; move to the rack
TRIGGER WHEN DISTANCE=1 DELAY=-1 DO Schrittmerker_R1Place(10310,10002,FPlace_R1_L4_S4_VP1,XPlace_R1_L4_S4_VP1) PRIO=-1
;FOLD PTP Place_R1_L4_S4_VP1 CONT Vel=12 % PPlace_R1_L4_S4_VP1 Tool[2]:Lower Gripper Base[0];%{PE}%R8.3.21,%MKUKATPBASIS,%CMOVE,%VPTP,%P 1:PTP, 2:Place_R1_L4_S4_VP1, 3:C_DIS, 5:12, 7:PPlace_R1_L4_S4_VP1
$BWDSTART=FALSE
PDAT_ACT= PPPlace_R1_L4_S4_VP1
FDAT_ACT= FPlace_R1_L4_S4_VP1
BAS(#PTP_PARAMS,12)
PTP XPlace_R1_L4_S4_VP1 C_DIS
;ENDFOLD
TRIGGER WHEN DISTANCE=1 DELAY=-1 DO Schrittmerker_R1Place(10311,10310,FPlace_R1_L4_S4_VP2,XPlace_R1_L4_S4_VP2) PRIO=-1
;FOLD PTP Place_R1_L4_S4_VP2 CONT Vel=12 % PPlace_R1_L4_S4_VP2 Tool[2]:Lower Gripper Base[0];%{PE}%R8.3.21,%MKUKATPBASIS,%CMOVE,%VPTP,%P 1:PTP, 2:Place_R1_L4_S4_VP2, 3:C_DIS, 5:12, 7:PPlace_R1_L4_S4_VP2
$BWDSTART=FALSE
PDAT_ACT= PPPlace_R1_L4_S4_VP2
FDAT_ACT= FPlace_R1_L4_S4_VP2
BAS(#PTP_PARAMS,12)
PTP XPlace_R1_L4_S4_VP2 C_DIS
;ENDFOLD
TRIGGER WHEN DISTANCE=1 DELAY=-1 DO Schrittmerker_R1Place(10312,10311,FPlace_R1_L4_S4_VP3,XPlace_R1_L4_S4_VP3) PRIO=-1
;FOLD PTP Place_R1_L4_S4_VP3 CONT Vel=12 % PPlace_R1_L4_S4_VP3 Tool[2]:Lower Gripper Base[1]:Rack1;%{PE}%R8.3.21,%MKUKATPBASIS,%CMOVE,%VPTP,%P 1:PTP, 2:Place_R1_L4_S4_VP3, 3:C_DIS, 5:12, 7:PPlace_R1_L4_S4_VP3
$BWDSTART=FALSE
PDAT_ACT= PPPlace_R1_L4_S4_VP3
FDAT_ACT= FPlace_R1_L4_S4_VP3
BAS(#PTP_PARAMS,12)
PTP XPlace_R1_L4_S4_VP3 C_DIS
;ENDFOLD

TRIGGER WHEN DISTANCE=1 DELAY=-1 DO Schrittmerker_R1Place(10313,10312,FPlace_R1_L4_S4_Check,XPlace_R1_L4_S4_Check) PRIO=-1
;FOLD PTP Place_R1_L4_S4_Check Vel=12 % PPlace_R1_L4_S4_Check Tool[2]:Lower Gripper Base[1]:Rack1;%{PE}%R8.3.21,%MKUKATPBASIS,%CMOVE,%VPTP,%P 1:PTP, 2:Place_R1_L4_S4_Check, 3:, 5:12, 7:PPlace_R1_L4_S4_Check
$BWDSTART=FALSE
PDAT_ACT= PPPlace_R1_L4_S4_Check
FDAT_ACT= FPlace_R1_L4_S4_Check
BAS(#PTP_PARAMS,12)
PTP XPlace_R1_L4_S4_Check
;ENDFOLD

;***************************************************
;FOLD Pruefe Platz frei
IF (DetectPart(CHECK_SHELF,PLACE)==OCCUPIED) THEN
  UP_Rueckzug_R1Place( )
  RETURN
ENDIF
;ENDFOLD
;***************************************************

TRIGGER WHEN DISTANCE=1 DELAY=-1 DO Schrittmerker_R1Place(10314,10313,FPlace_R1_L4_S4_VP4,XPlace_R1_L4_S4_VP4) PRIO=-1
;FOLD LIN Place_R1_L4_S4_VP4 CONT Vel=0.5 m/s LPlace_R1_L4_S4_VP4 Tool[2]:Lower Gripper Base[1]:Rack1;%{PE}%R8.3.21,%MKUKATPBASIS,%CMOVE,%VLIN,%P 1:LIN, 2:Place_R1_L4_S4_VP4, 3:C_DIS C_DIS, 5:0.5, 7:LPlace_R1_L4_S4_VP4
$BWDSTART=FALSE
LDAT_ACT= LLPlace_R1_L4_S4_VP4
FDAT_ACT= FPlace_R1_L4_S4_VP4
BAS(#CP_PARAMS,0.5)
LIN XPlace_R1_L4_S4_VP4 C_DIS C_DIS
;ENDFOLD
TRIGGER WHEN DISTANCE=1 DELAY=-1 DO Schrittmerker_R1Place(10315,10314,FPlace_R1_L4_S4_VP5,XPlace_R1_L4_S4_VP5) PRIO=-1
;FOLD LIN Place_R1_L4_S4_VP5 CONT Vel=0.5 m/s LPlace_R1_L4_S4_VP5 Tool[2]:Lower Gripper Base[1]:Rack1;%{PE}%R8.3.21,%MKUKATPBASIS,%CMOVE,%VLIN,%P 1:LIN, 2:Place_R1_L4_S4_VP5, 3:C_DIS C_DIS, 5:0.5, 7:LPlace_R1_L4_S4_VP5
$BWDSTART=FALSE
LDAT_ACT= LLPlace_R1_L4_S4_VP5
FDAT_ACT= FPlace_R1_L4_S4_VP5
BAS(#CP_PARAMS,0.5)
LIN XPlace_R1_L4_S4_VP5 C_DIS C_DIS
;ENDFOLD

;FOLD Test the way back home - part 1
CONTINUE
IF ($FLAG[M_Test_GrdstFahren1] AND NOT $FLAG[M_Test_GrdstFahren2]) THEN
  $FLAG[M_Test_GrdstFahren2]=TRUE
  UP_Rueckzug( )
  RETURN
ENDIF
;ENDFOLD

;-------------------------------
; Place part position
;-------------------------------
TRIGGER WHEN DISTANCE=1 DELAY=-1 DO Schrittmerker_R1Place(10316,10317,FPlace_R1_L4_S4_AP,XPlace_R1_L4_S4_AP) PRIO=-1
;FOLD LIN Place_R1_L4_S4_AP Vel=0.2 m/s LPlace_R1_L4_S4_AP Tool[2]:Lower Gripper Base[1]:Rack1;%{PE}%R8.3.21,%MKUKATPBASIS,%CMOVE,%VLIN,%P 1:LIN, 2:Place_R1_L4_S4_AP, 3:, 5:0.2, 7:LPlace_R1_L4_S4_AP
$BWDSTART=FALSE
LDAT_ACT= LLPlace_R1_L4_S4_AP
FDAT_ACT= FPlace_R1_L4_S4_AP
BAS(#CP_PARAMS,0.2)
LIN XPlace_R1_L4_S4_AP
;ENDFOLD

;FOLD Test the way back home - part 2
CONTINUE
IF $FLAG[M_Test_GrdstFahren2] THEN
  $FLAG[M_Test_GrdstFahren2]=FALSE
  UP_Rueckzug( )
  RETURN
ENDIF
;ENDFOLD

;***************************************************
; Disable part lost detection
SetPartLostDetection(NO_PART)
;***************************************************

TRIGGER WHEN DISTANCE=1 DELAY=-1 DO Schrittmerker_R1Place(10317,10318,FPlace_R1_L4_S4_NP1,XPlace_R1_L4_S4_NP1) PRIO=-1
;FOLD LIN Place_R1_L4_S4_NP1 Vel=0.2 m/s LPlace_R1_L4_S4_NP1 Tool[2]:Lower Gripper Base[1]:Rack1;%{PE}%R8.3.21,%MKUKATPBASIS,%CMOVE,%VLIN,%P 1:LIN, 2:Place_R1_L4_S4_NP1, 3:C_DIS C_DIS, 5:0.2, 7:LPlace_R1_L4_S4_NP1
$BWDSTART=FALSE
LDAT_ACT= LLPlace_R1_L4_S4_NP1
FDAT_ACT= FPlace_R1_L4_S4_NP1
BAS(#CP_PARAMS,0.2)
LIN XPlace_R1_L4_S4_NP1
;ENDFOLD

;***************************************************
; Check for part present (empty gripper)
CheckPartPresent(EMPTY_GRIPPER)
;***************************************************
; set load data
SetLoadData( )
;***************************************************

TRIGGER WHEN DISTANCE=1 DELAY=-1 DO Schrittmerker_R1Place(10318,10319,FPlace_R1_L4_S4_NP2,XPlace_R1_L4_S4_NP2) PRIO=-1
;FOLD LIN Place_R1_L4_S4_NP2 CONT Vel=0.5 m/s LPlace_R1_L4_S4_NP2 Tool[2]:Lower Gripper Base[1]:Rack1;%{PE}%R8.3.21,%MKUKATPBASIS,%CMOVE,%VLIN,%P 1:LIN, 2:Place_R1_L4_S4_NP2, 3:C_DIS C_DIS, 5:0.5, 7:LPlace_R1_L4_S4_NP2
$BWDSTART=FALSE
LDAT_ACT= LLPlace_R1_L4_S4_NP2
FDAT_ACT= FPlace_R1_L4_S4_NP2
BAS(#CP_PARAMS,0.5)
LIN XPlace_R1_L4_S4_NP2 C_DIS C_DIS
;ENDFOLD
TRIGGER WHEN DISTANCE=1 DELAY=-1 DO Schrittmerker_R1Place(10319,10320,FPlace_R1_L4_S4_NP3,XPlace_R1_L4_S4_NP3) PRIO=-1
;FOLD LIN Place_R1_L4_S4_NP3 Vel=0.5 m/s LPlace_R1_L4_S4_NP3 Tool[2]:Lower Gripper Base[1]:Rack 1 ;%{PE}
$BWDSTART=FALSE
LDAT_ACT= LLPlace_R1_L4_S4_NP3
FDAT_ACT= FPlace_R1_L4_S4_NP3
BAS(#CP_PARAMS,0.5)
LIN XPlace_R1_L4_S4_NP3
;ENDFOLD
TRIGGER WHEN DISTANCE=1 DELAY=-1 DO Schrittmerker_R1Place(10320,10321,FPlace_R1_L4_S4_NP4,XPlace_R1_L4_S4_NP4) PRIO=-1
;FOLD PTP Place_R1_L4_S4_NP4 CONT Vel=100 % PPlace_R1_L4_S4_NP4 Tool[2]:Lower Gripper Base[0];%{PE}%R8.3.21,%MKUKATPBASIS,%CMOVE,%VPTP,%P 1:PTP, 2:Place_R1_L4_S4_NP4, 3:C_DIS, 5:100, 7:PPlace_R1_L4_S4_NP4
$BWDSTART=FALSE
PDAT_ACT= PPPlace_R1_L4_S4_NP4
FDAT_ACT= FPlace_R1_L4_S4_NP4
BAS(#PTP_PARAMS,100)
PTP XPlace_R1_L4_S4_NP4 C_DIS
;ENDFOLD
TRIGGER WHEN DISTANCE=1 DELAY=-1 DO Schrittmerker_R1Place(10321,10322,FPlace_R1_L4_S4_NP5,XPlace_R1_L4_S4_NP5) PRIO=-1
;FOLD PTP Place_R1_L4_S4_NP5 CONT Vel=100 % PPlace_R1_L4_S4_NP5 Tool[2]:Lower Gripper Base[0];%{PE}%R8.3.21,%MKUKATPBASIS,%CMOVE,%VPTP,%P 1:PTP, 2:Place_R1_L4_S4_NP5, 3:C_DIS, 5:100, 7:PPlace_R1_L4_S4_NP5
$BWDSTART=FALSE
PDAT_ACT= PPPlace_R1_L4_S4_NP5
FDAT_ACT= FPlace_R1_L4_S4_NP5
BAS(#PTP_PARAMS,100)
PTP XPlace_R1_L4_S4_NP5 C_DIS
;ENDFOLD
TRIGGER WHEN DISTANCE=1 DELAY=-1 DO Schrittmerker_R1Place(10322,10323,FPlace_R1_L4_S4_NP6,XPlace_R1_L4_S4_NP6) PRIO=-1
;FOLD PTP Place_R1_L4_S4_NP6 CONT Vel=100 % PPlace_R1_L4_S4_NP6 Tool[2]:Lower Gripper Base[0];%{PE}%R8.3.21,%MKUKATPBASIS,%CMOVE,%VPTP,%P 1:PTP, 2:Place_R1_L4_S4_NP6, 3:C_DIS, 5:100, 7:PPlace_R1_L4_S4_NP6
$BWDSTART=FALSE
PDAT_ACT= PPPlace_R1_L4_S4_NP6
FDAT_ACT= FPlace_R1_L4_S4_NP6
BAS(#PTP_PARAMS,100)
PTP XPlace_R1_L4_S4_NP6 C_DIS
;ENDFOLD

TRIGGER WHEN DISTANCE=1 DELAY=-1 DO Schrittmerker_R1Place(10323,10002,FHOME1,$nullframe,XHOME1) PRIO=-1
;FOLD PTP HOME1 Vel=100 % PHome1;%{PE}%R8.3.21,%MKUKATPBASIS,%CMOVE,%VPTP,%P 1:PTP, 2:HOME1, 3:, 5:100, 7:PHome1
$BWDSTART=FALSE
PDAT_ACT= PPHome1
FDAT_ACT= FHOME1
BAS(#PTP_PARAMS,100)
PTP XHOME1
;ENDFOLD

;***************************************************
;FOLD Final tasks.
; Robot out of area Rack 1 Level 4
RobAusStorage1_4_A70=RESET_IN_AREA
;***************************************************
; stop cyclic clearence check
$CYCFLAG[ciFreigabeSPS]=DISABLE_MONITORING
;***************************************************
; Disable collision detection
;FOLD COLLDETECT Off ;%{PE}
;FOLD Parameters ;%{h}
;Params IlfProvider=kukaroboter.basistech.inlineforms.colldetect.off; CollDetect.Command=Off
;ENDFOLD
USE_CD_PARAMS(0)
;ENDFOLD
;***************************************************
;ENDFOLD
;***************************************************

END

; ##################################################

GLOBAL DEF UP_Place_R1_L5_S1( )
;***************************************************
; Place part on:
;    Rack  1
;    Level 5
;    Shelf 1
;***************************************************
;FOLD Preconditions - Vorraussetzungen
;***************************************************
; Enable collision detection
;FOLD COLLDETECT SetLimits Axis1: 150 % Axis2: 200 % Axis3: 150 % Axis4: 200 % Axis5: 150 % Axis6: 150 % ;%{PE}
;FOLD Parameters ;%{h}
;Params IlfProvider=kukaroboter.basistech.inlineforms.colldetect.setlimits; CollDetect.Command=SetLimits; CollDetect.Axis1=150; CollDetect.Axis2=200; CollDetect.Axis3=150; CollDetect.Axis4=200; CollDetect.Axis5=150; CollDetect.Axis6=150
;ENDFOLD
SET_TQ_VALUES(150, 200, 150, 200, 150, 150)
;ENDFOLD
;***************************************************
; Check for part in gripper (tool 1).
CheckPartPresent(OCCUPIED_GRIPPER,PART_ON_TOOL_1)
;***************************************************
; Enable part lost detection for tool 1
SetPartLostDetection(PART_ON_TOOL_1)
;***************************************************
; Set load data.
SetLoadData( )
;***************************************************
; Robot has to start from home position.
IF NOT $IN_HOME THEN
  UP_HomeToHome(0)
ENDIF
;***************************************************
;ENDFOLD

TRIGGER WHEN DISTANCE=1 DELAY=-1 DO Schrittmerker_R1Place(10501,10501,FHOME,$nullframe,XHOME) PRIO=-1
;FOLD PTP HOME Vel=12 % PHome;%{PE}%R8.3.21,%MKUKATPBASIS,%CMOVE,%VPTP,%P 1:PTP, 2:HOME, 3:, 5:12, 7:PHome
$BWDSTART=FALSE
PDAT_ACT= PPHome
FDAT_ACT= FHOME
BAS(#PTP_PARAMS,12)
PTP XHOME
;ENDFOLD

;***************************************************
;FOLD Area clearence handshake.
IF NOT $FLAG[M_Inbetriebnahme] THEN
  ;-------------------------------------------------
  ; Request area clearence.
  AnfStoer_Store1_5_A103=SET_REQUEST
  ;-------------------------------------------------
  ; Wait for area clearence from PLC.
  WAIT_FOR_INPUT("Frg_Storage1_5_E71",TRUE)
  ;-------------------------------------------------
  ; Reset area clearence request.
  AnfStoer_Store1_5_A103=RESET_REQUEST
  ;-------------------------------------------------
  ; start cyclic clearence check
  $CYCFLAG[ciFreigabeSPS]=Frg_Storage1_5_E71
  ;-------------------------------------------------
ENDIF
;***************************************************
; set "robot in area"
RobAusStorage1_5_A71=SET_IN_AREA
;ENDFOLD
;***************************************************

;***************************************************
;FOLD Check for Teachmode
IF $FLAG[M_Teachen] THEN
  WAIT FOR $T1
ENDIF
;ENDFOLD
;***************************************************

; move to the rack
TRIGGER WHEN DISTANCE=1 DELAY=-1 DO Schrittmerker_R1Place(10510,10501,FPlace_R1_L5_S1_VP1,XPlace_R1_L5_S1_VP1) PRIO=-1
;FOLD PTP Place_R1_L5_S1_VP1 CONT Vel=12 % PPlace_R1_L5_S1_VP1 Tool[1]:Upper Gripper Base[0];%{PE}%R8.3.21,%MKUKATPBASIS,%CMOVE,%VPTP,%P 1:PTP, 2:Place_R1_L5_S1_VP1, 3:C_DIS, 5:12, 7:PPlace_R1_L5_S1_VP1
$BWDSTART=FALSE
PDAT_ACT= PPPlace_R1_L5_S1_VP1
FDAT_ACT= FPlace_R1_L5_S1_VP1
BAS(#PTP_PARAMS,12)
PTP XPlace_R1_L5_S1_VP1 C_DIS
;ENDFOLD
TRIGGER WHEN DISTANCE=1 DELAY=-1 DO Schrittmerker_R1Place(10511,10510,FPlace_R1_L5_S1_VP2,XPlace_R1_L5_S1_VP2) PRIO=-1
;FOLD PTP Place_R1_L5_S1_VP2 CONT Vel=12 % PPlace_R1_L5_S1_VP2 Tool[1]:Upper Gripper Base[0];%{PE}%R8.3.21,%MKUKATPBASIS,%CMOVE,%VPTP,%P 1:PTP, 2:Place_R1_L5_S1_VP2, 3:C_DIS, 5:12, 7:PPlace_R1_L5_S1_VP2
$BWDSTART=FALSE
PDAT_ACT= PPPlace_R1_L5_S1_VP2
FDAT_ACT= FPlace_R1_L5_S1_VP2
BAS(#PTP_PARAMS,12)
PTP XPlace_R1_L5_S1_VP2 C_DIS
;ENDFOLD
TRIGGER WHEN DISTANCE=1 DELAY=-1 DO Schrittmerker_R1Place(10512,10511,FPlace_R1_L5_S1_VP3,XPlace_R1_L5_S1_VP3) PRIO=-1
;FOLD PTP Place_R1_L5_S1_VP3 CONT Vel=12 % PPlace_R1_L5_S1_VP3 Tool[1]:Upper Gripper Base[0];%{PE}%R8.3.21,%MKUKATPBASIS,%CMOVE,%VPTP,%P 1:PTP, 2:Place_R1_L5_S1_VP3, 3:C_DIS, 5:12, 7:PPlace_R1_L5_S1_VP3
$BWDSTART=FALSE
PDAT_ACT= PPPlace_R1_L5_S1_VP3
FDAT_ACT= FPlace_R1_L5_S1_VP3
BAS(#PTP_PARAMS,12)
PTP XPlace_R1_L5_S1_VP3 C_DIS
;ENDFOLD
TRIGGER WHEN DISTANCE=1 DELAY=-1 DO Schrittmerker_R1Place(10513,10512,FPlace_R1_L5_S1_VP4,XPlace_R1_L5_S1_VP4) PRIO=-1
;FOLD PTP Place_R1_L5_S1_VP4 CONT Vel=12 % PPlace_R1_L5_S1_VP4 Tool[1]:Upper Gripper Base[0];%{PE}%R8.3.21,%MKUKATPBASIS,%CMOVE,%VPTP,%P 1:PTP, 2:Place_R1_L5_S1_VP4, 3:C_DIS, 5:12, 7:PPlace_R1_L5_S1_VP4
$BWDSTART=FALSE
PDAT_ACT= PPPlace_R1_L5_S1_VP4
FDAT_ACT= FPlace_R1_L5_S1_VP4
BAS(#PTP_PARAMS,12)
PTP XPlace_R1_L5_S1_VP4 C_DIS
;ENDFOLD
TRIGGER WHEN DISTANCE=1 DELAY=-1 DO Schrittmerker_R1Place(10514,10513,FPlace_R1_L5_S1_VP5,XPlace_R1_L5_S1_VP5) PRIO=-1
;FOLD PTP Place_R1_L5_S1_VP5 CONT Vel=12 % PPlace_R1_L5_S1_VP5 Tool[1]:Upper Gripper Base[0];%{PE}%R8.3.21,%MKUKATPBASIS,%CMOVE,%VPTP,%P 1:PTP, 2:Place_R1_L5_S1_VP5, 3:C_DIS, 5:12, 7:PPlace_R1_L5_S1_VP5
$BWDSTART=FALSE
PDAT_ACT= PPPlace_R1_L5_S1_VP5
FDAT_ACT= FPlace_R1_L5_S1_VP5
BAS(#PTP_PARAMS,12)
PTP XPlace_R1_L5_S1_VP5 C_DIS
;ENDFOLD
TRIGGER WHEN DISTANCE=1 DELAY=-1 DO Schrittmerker_R1Place(10515,10514,FPlace_R1_L5_S1_VP6,XPlace_R1_L5_S1_VP6) PRIO=-1
;FOLD PTP Place_R1_L5_S1_VP6 CONT Vel=12 % PPlace_R1_L5_S1_VP6 Tool[1]:Upper Gripper Base[0];%{PE}%R8.3.21,%MKUKATPBASIS,%CMOVE,%VPTP,%P 1:PTP, 2:Place_R1_L5_S1_VP6, 3:C_DIS, 5:12, 7:PPlace_R1_L5_S1_VP6
$BWDSTART=FALSE
PDAT_ACT= PPPlace_R1_L5_S1_VP6
FDAT_ACT= FPlace_R1_L5_S1_VP6
BAS(#PTP_PARAMS,12)
PTP XPlace_R1_L5_S1_VP6 C_DIS
;ENDFOLD
TRIGGER WHEN DISTANCE=1 DELAY=-1 DO Schrittmerker_R1Place(10516,10515,FPlace_R1_L5_S1_VP7,XPlace_R1_L5_S1_VP7) PRIO=-1
;FOLD PTP Place_R1_L5_S1_VP7 CONT Vel=12 % PPlace_R1_L5_S1_VP7 Tool[1]:Upper Gripper Base[0];%{PE}%R8.3.21,%MKUKATPBASIS,%CMOVE,%VPTP,%P 1:PTP, 2:Place_R1_L5_S1_VP7, 3:C_DIS, 5:12, 7:PPlace_R1_L5_S1_VP7
$BWDSTART=FALSE
PDAT_ACT= PPPlace_R1_L5_S1_VP7
FDAT_ACT= FPlace_R1_L5_S1_VP7
BAS(#PTP_PARAMS,12)
PTP XPlace_R1_L5_S1_VP7 C_DIS
;ENDFOLD
TRIGGER WHEN DISTANCE=1 DELAY=-1 DO Schrittmerker_R1Place(10517,10516,FPlace_R1_L5_S1_VP8,XPlace_R1_L5_S1_VP8) PRIO=-1
;FOLD PTP Place_R1_L5_S1_VP8 CONT Vel=12 % PPlace_R1_L5_S1_VP8 Tool[1]:Upper Gripper Base[0];%{PE}%R8.3.21,%MKUKATPBASIS,%CMOVE,%VPTP,%P 1:PTP, 2:Place_R1_L5_S1_VP8, 3:C_DIS, 5:12, 7:PPlace_R1_L5_S1_VP8
$BWDSTART=FALSE
PDAT_ACT= PPPlace_R1_L5_S1_VP8
FDAT_ACT= FPlace_R1_L5_S1_VP8
BAS(#PTP_PARAMS,12)
PTP XPlace_R1_L5_S1_VP8 C_DIS
;ENDFOLD
TRIGGER WHEN DISTANCE=1 DELAY=-1 DO Schrittmerker_R1Place(10518,10517,FPlace_R1_L5_S1_VP9,XPlace_R1_L5_S1_VP9) PRIO=-1
;FOLD PTP Place_R1_L5_S1_VP9 CONT Vel=12 % PPlace_R1_L5_S1_VP9 Tool[1]:Upper Gripper Base[1]:Rack1;%{PE}%R8.3.21,%MKUKATPBASIS,%CMOVE,%VPTP,%P 1:PTP, 2:Place_R1_L5_S1_VP9, 3:C_DIS, 5:12, 7:PPlace_R1_L5_S1_VP9
$BWDSTART=FALSE
PDAT_ACT= PPPlace_R1_L5_S1_VP9
FDAT_ACT= FPlace_R1_L5_S1_VP9
BAS(#PTP_PARAMS,12)
PTP XPlace_R1_L5_S1_VP9 C_DIS
;ENDFOLD
TRIGGER WHEN DISTANCE=1 DELAY=-1 DO Schrittmerker_R1Place(10519,10518,FPlace_R1_L5_S1_VP10,XPlace_R1_L5_S1_VP10) PRIO=-1
;FOLD PTP Place_R1_L5_S1_VP10 CONT Vel=12 % PPlace_R1_L5_S1_VP10 Tool[1]:Upper Gripper Base[1]:Rack1;%{PE}%R8.3.21,%MKUKATPBASIS,%CMOVE,%VPTP,%P 1:PTP, 2:Place_R1_L5_S1_VP10, 3:C_DIS, 5:12, 7:PPlace_R1_L5_S1_VP10
$BWDSTART=FALSE
PDAT_ACT= PPPlace_R1_L5_S1_VP10
FDAT_ACT= FPlace_R1_L5_S1_VP10
BAS(#PTP_PARAMS,12)
PTP XPlace_R1_L5_S1_VP10 C_DIS
;ENDFOLD

TRIGGER WHEN DISTANCE=1 DELAY=-1 DO Schrittmerker_R1Place(10520,10519,FPlace_R1_L5_S1_Check,XPlace_R1_L5_S1_Check) PRIO=-1
;FOLD PTP Place_R1_L5_S1_Check Vel=12 % PPlace_R1_L5_S1_Check Tool[1]:Upper Gripper Base[1]:Rack1;%{PE}%R8.3.21,%MKUKATPBASIS,%CMOVE,%VPTP,%P 1:PTP, 2:Place_R1_L5_S1_Check, 3:, 5:12, 7:PPlace_R1_L5_S1_Check
$BWDSTART=FALSE
PDAT_ACT= PPPlace_R1_L5_S1_Check
FDAT_ACT= FPlace_R1_L5_S1_Check
BAS(#PTP_PARAMS,12)
PTP XPlace_R1_L5_S1_Check
;ENDFOLD

;***************************************************
;FOLD Pruefe Platz frei
IF (DetectPart(CHECK_SHELF,PLACE)==OCCUPIED) THEN
  UP_Rueckzug_R1Place( )
  RETURN
ENDIF
;ENDFOLD
;***************************************************

TRIGGER WHEN DISTANCE=1 DELAY=-1 DO Schrittmerker_R1Place(10521,10520,FPlace_R1_L5_S1_VP11,XPlace_R1_L5_S1_VP11) PRIO=-1
;FOLD LIN Place_R1_L5_S1_VP11 CONT Vel=0.5 m/s LPlace_R1_L5_S1_VP11 Tool[1]:Upper Gripper Base[1]:Rack1;%{PE}%R8.3.21,%MKUKATPBASIS,%CMOVE,%VLIN,%P 1:LIN, 2:Place_R1_L5_S1_VP11, 3:C_DIS C_DIS, 5:0.5, 7:LPlace_R1_L5_S1_VP11
$BWDSTART=FALSE
LDAT_ACT= LLPlace_R1_L5_S1_VP11
FDAT_ACT= FPlace_R1_L5_S1_VP11
BAS(#CP_PARAMS,0.5)
LIN XPlace_R1_L5_S1_VP11 C_DIS C_DIS
;ENDFOLD

;FOLD Test the way back home - part 1
CONTINUE
IF ($FLAG[M_Test_GrdstFahren1] AND NOT $FLAG[M_Test_GrdstFahren2]) THEN
  $FLAG[M_Test_GrdstFahren2]=TRUE
  UP_Rueckzug( )
  RETURN
ENDIF
;ENDFOLD

;-------------------------------
; Place part position
;-------------------------------
TRIGGER WHEN DISTANCE=1 DELAY=-1 DO Schrittmerker_R1Place(10522,10523,FPlace_R1_L5_S1_AP,XPlace_R1_L5_S1_AP) PRIO=-1
;FOLD LIN Place_R1_L5_S1_AP Vel=0.2 m/s LPlace_R1_L5_S1_AP Tool[1]:Upper Gripper Base[1]:Rack1;%{PE}%R8.3.21,%MKUKATPBASIS,%CMOVE,%VLIN,%P 1:LIN, 2:Place_R1_L5_S1_AP, 3:, 5:0.2, 7:LPlace_R1_L5_S1_AP
$BWDSTART=FALSE
LDAT_ACT= LLPlace_R1_L5_S1_AP
FDAT_ACT= FPlace_R1_L5_S1_AP
BAS(#CP_PARAMS,0.2)
LIN XPlace_R1_L5_S1_AP
;ENDFOLD

;FOLD Test the way back home - part 2
CONTINUE
IF $FLAG[M_Test_GrdstFahren2] THEN
  $FLAG[M_Test_GrdstFahren2]=FALSE
  UP_Rueckzug( )
  RETURN
ENDIF
;ENDFOLD

;***************************************************
; Disable part lost detection
SetPartLostDetection(NO_PART)
;***************************************************

TRIGGER WHEN DISTANCE=1 DELAY=-1 DO Schrittmerker_R1Place(10523,10524,FPlace_R1_L5_S1_NP1,XPlace_R1_L5_S1_NP1) PRIO=-1
;FOLD LIN Place_R1_L5_S1_NP1 Vel=0.2 m/s LPlace_R1_L5_S1_NP1 Tool[1]:Upper Gripper Base[1]:Rack1;%{PE}%R8.3.21,%MKUKATPBASIS,%CMOVE,%VLIN,%P 1:LIN, 2:Place_R1_L5_S1_NP1, 3:C_DIS C_DIS, 5:0.2, 7:LPlace_R1_L5_S1_NP1
$BWDSTART=FALSE
LDAT_ACT= LLPlace_R1_L5_S1_NP1
FDAT_ACT= FPlace_R1_L5_S1_NP1
BAS(#CP_PARAMS,0.2)
LIN XPlace_R1_L5_S1_NP1
;ENDFOLD

;***************************************************
; Check for part present (empty gripper)
CheckPartPresent(EMPTY_GRIPPER)
;***************************************************
; set load data
SetLoadData( )
;***************************************************

TRIGGER WHEN DISTANCE=1 DELAY=-1 DO Schrittmerker_R1Place(10524,10525,FPlace_R1_L5_S1_NP2,XPlace_R1_L5_S1_NP2) PRIO=-1
;FOLD LIN Place_R1_L5_S1_NP2 Vel=0.5 m/s LPlace_R1_L5_S1_NP2 Tool[1]:Upper Gripper Base[1]:Rack1;%{PE}%R8.3.21,%MKUKATPBASIS,%CMOVE,%VLIN,%P 1:LIN, 2:Place_R1_L5_S1_NP2, 3:, 5:0.5, 7:LPlace_R1_L5_S1_NP2
$BWDSTART=FALSE
LDAT_ACT= LLPlace_R1_L5_S1_NP2
FDAT_ACT= FPlace_R1_L5_S1_NP2
BAS(#CP_PARAMS,0.5)
LIN XPlace_R1_L5_S1_NP2
;ENDFOLD
TRIGGER WHEN DISTANCE=1 DELAY=-1 DO Schrittmerker_R1Place(10525,10526,FPlace_R1_L5_S1_NP3,XPlace_R1_L5_S1_NP3) PRIO=-1
;FOLD PTP Place_R1_L5_S1_NP3 CONT Vel=100 % PPlace_R1_L5_S1_NP3 Tool[1]:Upper Gripper Base[1]:Rack1;%{PE}%R8.3.21,%MKUKATPBASIS,%CMOVE,%VPTP,%P 1:PTP, 2:Place_R1_L5_S1_NP3, 3:C_DIS, 5:100, 7:PPlace_R1_L5_S1_NP3
$BWDSTART=FALSE
PDAT_ACT= PPPlace_R1_L5_S1_NP3
FDAT_ACT= FPlace_R1_L5_S1_NP3
BAS(#PTP_PARAMS,100)
PTP XPlace_R1_L5_S1_NP3 C_DIS
;ENDFOLD
TRIGGER WHEN DISTANCE=1 DELAY=-1 DO Schrittmerker_R1Place(10526,10527,FPlace_R1_L5_S1_NP4,XPlace_R1_L5_S1_NP4) PRIO=-1
;FOLD PTP Place_R1_L5_S1_NP4 CONT Vel=100 % PPlace_R1_L5_S1_NP4 Tool[1]:Upper Gripper Base[0];%{PE}%R8.3.21,%MKUKATPBASIS,%CMOVE,%VPTP,%P 1:PTP, 2:Place_R1_L5_S1_NP4, 3:C_DIS, 5:100, 7:PPlace_R1_L5_S1_NP4
$BWDSTART=FALSE
PDAT_ACT= PPPlace_R1_L5_S1_NP4
FDAT_ACT= FPlace_R1_L5_S1_NP4
BAS(#PTP_PARAMS,100)
PTP XPlace_R1_L5_S1_NP4 C_DIS
;ENDFOLD
TRIGGER WHEN DISTANCE=1 DELAY=-1 DO Schrittmerker_R1Place(10527,10528,FPlace_R1_L5_S1_NP5,XPlace_R1_L5_S1_NP5) PRIO=-1
;FOLD PTP Place_R1_L5_S1_NP5 CONT Vel=100 % PPlace_R1_L5_S1_NP5 Tool[1]:Upper Gripper Base[0];%{PE}%R8.3.21,%MKUKATPBASIS,%CMOVE,%VPTP,%P 1:PTP, 2:Place_R1_L5_S1_NP5, 3:C_DIS, 5:100, 7:PPlace_R1_L5_S1_NP5
$BWDSTART=FALSE
PDAT_ACT= PPPlace_R1_L5_S1_NP5
FDAT_ACT= FPlace_R1_L5_S1_NP5
BAS(#PTP_PARAMS,100)
PTP XPlace_R1_L5_S1_NP5 C_DIS
;ENDFOLD
TRIGGER WHEN DISTANCE=1 DELAY=-1 DO Schrittmerker_R1Place(10528,10529,FPlace_R1_L5_S1_NP6,XPlace_R1_L5_S1_NP6) PRIO=-1
;FOLD PTP Place_R1_L5_S1_NP6 CONT Vel=100 % PPlace_R1_L5_S1_NP6 Tool[1]:Upper Gripper Base[0];%{PE}%R8.3.21,%MKUKATPBASIS,%CMOVE,%VPTP,%P 1:PTP, 2:Place_R1_L5_S1_NP6, 3:C_DIS, 5:100, 7:PPlace_R1_L5_S1_NP6
$BWDSTART=FALSE
PDAT_ACT= PPPlace_R1_L5_S1_NP6
FDAT_ACT= FPlace_R1_L5_S1_NP6
BAS(#PTP_PARAMS,100)
PTP XPlace_R1_L5_S1_NP6 C_DIS
;ENDFOLD

TRIGGER WHEN DISTANCE=1 DELAY=-1 DO Schrittmerker_R1Place(10529,10501,FHOME,$nullframe,XHOME) PRIO=-1
;FOLD PTP HOME Vel=100 % PHome;%{PE}%R8.3.21,%MKUKATPBASIS,%CMOVE,%VPTP,%P 1:PTP, 2:HOME, 3:, 5:100, 7:PHome
$BWDSTART=FALSE
PDAT_ACT= PPHome
FDAT_ACT= FHOME
BAS(#PTP_PARAMS,100)
PTP XHOME
;ENDFOLD

;***************************************************
;FOLD Final tasks.
; Robot out of area Rack 1 Level 5
RobAusStorage1_5_A71=RESET_IN_AREA
;***************************************************
; stop cyclic clearence check
$CYCFLAG[ciFreigabeSPS]=DISABLE_MONITORING
;***************************************************
; Disable collision detection
;FOLD COLLDETECT Off ;%{PE}
;FOLD Parameters ;%{h}
;Params IlfProvider=kukaroboter.basistech.inlineforms.colldetect.off; CollDetect.Command=Off
;ENDFOLD
USE_CD_PARAMS(0)
;ENDFOLD
;***************************************************
;ENDFOLD
;***************************************************

END

; ##################################################

GLOBAL DEF UP_Place_R1_L5_S2( )
;***************************************************
; Place part on:
;    Rack  1
;    Level 5
;    Shelf 2
;***************************************************
;FOLD Preconditions - Vorraussetzungen
;***************************************************
; Enable collision detection
;FOLD COLLDETECT SetLimits Axis1: 150 % Axis2: 200 % Axis3: 150 % Axis4: 200 % Axis5: 150 % Axis6: 150 % ;%{PE}
;FOLD Parameters ;%{h}
;Params IlfProvider=kukaroboter.basistech.inlineforms.colldetect.setlimits; CollDetect.Command=SetLimits; CollDetect.Axis1=150; CollDetect.Axis2=200; CollDetect.Axis3=150; CollDetect.Axis4=200; CollDetect.Axis5=150; CollDetect.Axis6=150
;ENDFOLD
SET_TQ_VALUES(150, 200, 150, 200, 150, 150)
;ENDFOLD
;***************************************************
; Check for part in gripper (tool 1).
CheckPartPresent(OCCUPIED_GRIPPER,PART_ON_TOOL_1)
;***************************************************
; Enable part lost detection for tool 1
SetPartLostDetection(PART_ON_TOOL_1)
;***************************************************
; Set load data.
SetLoadData( )
;***************************************************
; Robot has to start from home position.
IF NOT $IN_HOME THEN
  UP_HomeToHome(0)
ENDIF
;***************************************************
;ENDFOLD

TRIGGER WHEN DISTANCE=1 DELAY=-1 DO Schrittmerker_R1Place(10501,10501,FHOME,$nullframe,XHOME) PRIO=-1
;FOLD PTP HOME Vel=12 % PHome;%{PE}%R8.3.21,%MKUKATPBASIS,%CMOVE,%VPTP,%P 1:PTP, 2:HOME, 3:, 5:12, 7:PHome
$BWDSTART=FALSE
PDAT_ACT= PPHome
FDAT_ACT= FHOME
BAS(#PTP_PARAMS,12)
PTP XHOME
;ENDFOLD

;***************************************************
;FOLD Area clearence handshake.
IF NOT $FLAG[M_Inbetriebnahme] THEN
  ;-------------------------------------------------
  ; Request area clearence.
  AnfStoer_Store1_5_A103=SET_REQUEST
  ;-------------------------------------------------
  ; Wait for area clearence from PLC.
  WAIT_FOR_INPUT("Frg_Storage1_5_E71",TRUE)
  ;-------------------------------------------------
  ; Reset area clearence request.
  AnfStoer_Store1_5_A103=RESET_REQUEST
  ;-------------------------------------------------
  ; start cyclic clearence check
  $CYCFLAG[ciFreigabeSPS]=Frg_Storage1_5_E71
  ;-------------------------------------------------
ENDIF
;***************************************************
; set "robot in area"
RobAusStorage1_5_A71=SET_IN_AREA
;ENDFOLD
;***************************************************

;***************************************************
;FOLD Check for Teachmode
IF $FLAG[M_Teachen] THEN
  WAIT FOR $T1
ENDIF
;ENDFOLD
;***************************************************

; move to the rack
TRIGGER WHEN DISTANCE=1 DELAY=-1 DO Schrittmerker_R1Place(10540,10501,FPlace_R1_L5_S2_VP1,XPlace_R1_L5_S2_VP1) PRIO=-1
;FOLD PTP Place_R1_L5_S2_VP1 CONT Vel=12 % PPlace_R1_L5_S2_VP1 Tool[1]:Upper Gripper Base[0];%{PE}%R8.3.21,%MKUKATPBASIS,%CMOVE,%VPTP,%P 1:PTP, 2:Place_R1_L5_S2_VP1, 3:C_DIS, 5:12, 7:PPlace_R1_L5_S2_VP1
$BWDSTART=FALSE
PDAT_ACT= PPPlace_R1_L5_S2_VP1
FDAT_ACT= FPlace_R1_L5_S2_VP1
BAS(#PTP_PARAMS,12)
PTP XPlace_R1_L5_S2_VP1 C_DIS
;ENDFOLD
TRIGGER WHEN DISTANCE=1 DELAY=-1 DO Schrittmerker_R1Place(10541,10540,FPlace_R1_L5_S2_VP2,XPlace_R1_L5_S2_VP2) PRIO=-1
;FOLD PTP Place_R1_L5_S2_VP2 CONT Vel=12 % PPlace_R1_L5_S2_VP2 Tool[1]:Upper Gripper Base[0];%{PE}%R8.3.21,%MKUKATPBASIS,%CMOVE,%VPTP,%P 1:PTP, 2:Place_R1_L5_S2_VP2, 3:C_DIS, 5:12, 7:PPlace_R1_L5_S2_VP2
$BWDSTART=FALSE
PDAT_ACT= PPPlace_R1_L5_S2_VP2
FDAT_ACT= FPlace_R1_L5_S2_VP2
BAS(#PTP_PARAMS,12)
PTP XPlace_R1_L5_S2_VP2 C_DIS
;ENDFOLD
TRIGGER WHEN DISTANCE=1 DELAY=-1 DO Schrittmerker_R1Place(10542,10541,FPlace_R1_L5_S2_VP3,XPlace_R1_L5_S2_VP3) PRIO=-1
;FOLD PTP Place_R1_L5_S2_VP3 CONT Vel=12 % PPlace_R1_L5_S2_VP3 Tool[1]:Upper Gripper Base[0];%{PE}%R8.3.21,%MKUKATPBASIS,%CMOVE,%VPTP,%P 1:PTP, 2:Place_R1_L5_S2_VP3, 3:C_DIS, 5:12, 7:PPlace_R1_L5_S2_VP3
$BWDSTART=FALSE
PDAT_ACT= PPPlace_R1_L5_S2_VP3
FDAT_ACT= FPlace_R1_L5_S2_VP3
BAS(#PTP_PARAMS,12)
PTP XPlace_R1_L5_S2_VP3 C_DIS
;ENDFOLD
TRIGGER WHEN DISTANCE=1 DELAY=-1 DO Schrittmerker_R1Place(10543,10542,FPlace_R1_L5_S2_VP4,XPlace_R1_L5_S2_VP4) PRIO=-1
;FOLD PTP Place_R1_L5_S2_VP4 CONT Vel=12 % PPlace_R1_L5_S2_VP4 Tool[1]:Upper Gripper Base[0];%{PE}%R8.3.21,%MKUKATPBASIS,%CMOVE,%VPTP,%P 1:PTP, 2:Place_R1_L5_S2_VP4, 3:C_DIS, 5:12, 7:PPlace_R1_L5_S2_VP4
$BWDSTART=FALSE
PDAT_ACT= PPPlace_R1_L5_S2_VP4
FDAT_ACT= FPlace_R1_L5_S2_VP4
BAS(#PTP_PARAMS,12)
PTP XPlace_R1_L5_S2_VP4 C_DIS
;ENDFOLD
TRIGGER WHEN DISTANCE=1 DELAY=-1 DO Schrittmerker_R1Place(10544,10543,FPlace_R1_L5_S2_VP5,XPlace_R1_L5_S2_VP5) PRIO=-1
;FOLD PTP Place_R1_L5_S2_VP5 CONT Vel=12 % PPlace_R1_L5_S2_VP5 Tool[1]:Upper Gripper Base[0];%{PE}%R8.3.21,%MKUKATPBASIS,%CMOVE,%VPTP,%P 1:PTP, 2:Place_R1_L5_S2_VP5, 3:C_DIS, 5:12, 7:PPlace_R1_L5_S2_VP5
$BWDSTART=FALSE
PDAT_ACT= PPPlace_R1_L5_S2_VP5
FDAT_ACT= FPlace_R1_L5_S2_VP5
BAS(#PTP_PARAMS,12)
PTP XPlace_R1_L5_S2_VP5 C_DIS
;ENDFOLD
TRIGGER WHEN DISTANCE=1 DELAY=-1 DO Schrittmerker_R1Place(10545,10544,FPlace_R1_L5_S2_VP6,XPlace_R1_L5_S2_VP6) PRIO=-1
;FOLD PTP Place_R1_L5_S2_VP6 CONT Vel=12 % PPlace_R1_L5_S2_VP6 Tool[1]:Upper Gripper Base[0];%{PE}%R8.3.21,%MKUKATPBASIS,%CMOVE,%VPTP,%P 1:PTP, 2:Place_R1_L5_S2_VP6, 3:C_DIS, 5:12, 7:PPlace_R1_L5_S2_VP6
$BWDSTART=FALSE
PDAT_ACT= PPPlace_R1_L5_S2_VP6
FDAT_ACT= FPlace_R1_L5_S2_VP6
BAS(#PTP_PARAMS,12)
PTP XPlace_R1_L5_S2_VP6 C_DIS
;ENDFOLD
TRIGGER WHEN DISTANCE=1 DELAY=-1 DO Schrittmerker_R1Place(10546,10545,FPlace_R1_L5_S2_VP7,XPlace_R1_L5_S2_VP7) PRIO=-1
;FOLD PTP Place_R1_L5_S2_VP7 CONT Vel=12 % PPlace_R1_L5_S2_VP7 Tool[1]:Upper Gripper Base[0];%{PE}%R8.3.21,%MKUKATPBASIS,%CMOVE,%VPTP,%P 1:PTP, 2:Place_R1_L5_S2_VP7, 3:C_DIS, 5:12, 7:PPlace_R1_L5_S2_VP7
$BWDSTART=FALSE
PDAT_ACT= PPPlace_R1_L5_S2_VP7
FDAT_ACT= FPlace_R1_L5_S2_VP7
BAS(#PTP_PARAMS,12)
PTP XPlace_R1_L5_S2_VP7 C_DIS
;ENDFOLD
TRIGGER WHEN DISTANCE=1 DELAY=-1 DO Schrittmerker_R1Place(10547,10546,FPlace_R1_L5_S2_VP8,XPlace_R1_L5_S2_VP8) PRIO=-1
;FOLD PTP Place_R1_L5_S2_VP8 CONT Vel=12 % PPlace_R1_L5_S2_VP8 Tool[1]:Upper Gripper Base[0];%{PE}%R8.3.21,%MKUKATPBASIS,%CMOVE,%VPTP,%P 1:PTP, 2:Place_R1_L5_S2_VP8, 3:C_DIS, 5:12, 7:PPlace_R1_L5_S2_VP8
$BWDSTART=FALSE
PDAT_ACT= PPPlace_R1_L5_S2_VP8
FDAT_ACT= FPlace_R1_L5_S2_VP8
BAS(#PTP_PARAMS,12)
PTP XPlace_R1_L5_S2_VP8 C_DIS
;ENDFOLD
TRIGGER WHEN DISTANCE=1 DELAY=-1 DO Schrittmerker_R1Place(10548,10547,FPlace_R1_L5_S2_VP9,XPlace_R1_L5_S2_VP9) PRIO=-1
;FOLD PTP Place_R1_L5_S2_VP9 CONT Vel=12 % PPlace_R1_L5_S2_VP9 Tool[1]:Upper Gripper Base[1]:Rack1;%{PE}%R8.3.21,%MKUKATPBASIS,%CMOVE,%VPTP,%P 1:PTP, 2:Place_R1_L5_S2_VP9, 3:C_DIS, 5:12, 7:PPlace_R1_L5_S2_VP9
$BWDSTART=FALSE
PDAT_ACT= PPPlace_R1_L5_S2_VP9
FDAT_ACT= FPlace_R1_L5_S2_VP9
BAS(#PTP_PARAMS,12)
PTP XPlace_R1_L5_S2_VP9 C_DIS
;ENDFOLD

TRIGGER WHEN DISTANCE=1 DELAY=-1 DO Schrittmerker_R1Place(10549,10548,FPlace_R1_L5_S2_Check,XPlace_R1_L5_S2_Check) PRIO=-1
;FOLD PTP Place_R1_L5_S2_Check Vel=12 % PPlace_R1_L5_S2_Check Tool[1]:Upper Gripper Base[1]:Rack1;%{PE}%R8.3.21,%MKUKATPBASIS,%CMOVE,%VPTP,%P 1:PTP, 2:Place_R1_L5_S2_Check, 3:, 5:12, 7:PPlace_R1_L5_S2_Check
$BWDSTART=FALSE
PDAT_ACT= PPPlace_R1_L5_S2_Check
FDAT_ACT= FPlace_R1_L5_S2_Check
BAS(#PTP_PARAMS,12)
PTP XPlace_R1_L5_S2_Check
;ENDFOLD

;***************************************************
;FOLD Pruefe Platz frei
IF (DetectPart(CHECK_SHELF,PLACE)==OCCUPIED) THEN
  UP_Rueckzug_R1Place( )
  RETURN
ENDIF
;ENDFOLD
;***************************************************

TRIGGER WHEN DISTANCE=1 DELAY=-1 DO Schrittmerker_R1Place(10550,10549,FPlace_R1_L5_S2_VP10,XPlace_R1_L5_S2_VP10) PRIO=-1
;FOLD LIN Place_R1_L5_S2_VP10 CONT Vel=0.5 m/s LPlace_R1_L5_S2_VP10 Tool[1]:Upper Gripper Base[1]:Rack1;%{PE}%R8.3.21,%MKUKATPBASIS,%CMOVE,%VLIN,%P 1:LIN, 2:Place_R1_L5_S2_VP10, 3:C_DIS C_DIS, 5:0.5, 7:LPlace_R1_L5_S2_VP10
$BWDSTART=FALSE
LDAT_ACT= LLPlace_R1_L5_S2_VP10
FDAT_ACT= FPlace_R1_L5_S2_VP10
BAS(#CP_PARAMS,0.5)
LIN XPlace_R1_L5_S2_VP10 C_DIS C_DIS
;ENDFOLD
TRIGGER WHEN DISTANCE=1 DELAY=-1 DO Schrittmerker_R1Place(10551,10550,FPlace_R1_L5_S2_VP11,XPlace_R1_L5_S2_VP11) PRIO=-1
;FOLD LIN Place_R1_L5_S2_VP11 CONT Vel=0.5 m/s LPlace_R1_L5_S2_VP11 Tool[1]:Upper Gripper Base[1]:Rack1;%{PE}%R8.3.21,%MKUKATPBASIS,%CMOVE,%VLIN,%P 1:LIN, 2:Place_R1_L5_S2_VP11, 3:C_DIS C_DIS, 5:0.5, 7:LPlace_R1_L5_S2_VP11
$BWDSTART=FALSE
LDAT_ACT= LLPlace_R1_L5_S2_VP11
FDAT_ACT= FPlace_R1_L5_S2_VP11
BAS(#CP_PARAMS,0.5)
LIN XPlace_R1_L5_S2_VP11 C_DIS C_DIS
;ENDFOLD
TRIGGER WHEN DISTANCE=1 DELAY=-1 DO Schrittmerker_R1Place(10552,10551,FPlace_R1_L5_S2_VP12,XPlace_R1_L5_S2_VP12) PRIO=-1
;FOLD LIN Place_R1_L5_S2_VP12 CONT Vel=0.5 m/s LPlace_R1_L5_S2_VP12 Tool[1]:Upper Gripper Base[1]:Rack1;%{PE}%R8.3.21,%MKUKATPBASIS,%CMOVE,%VLIN,%P 1:LIN, 2:Place_R1_L5_S2_VP12, 3:C_DIS C_DIS, 5:0.5, 7:LPlace_R1_L5_S2_VP12
$BWDSTART=FALSE
LDAT_ACT= LLPlace_R1_L5_S2_VP12
FDAT_ACT= FPlace_R1_L5_S2_VP12
BAS(#CP_PARAMS,0.5)
LIN XPlace_R1_L5_S2_VP12 C_DIS C_DIS
;ENDFOLD

;FOLD Test the way back home - part 1
CONTINUE
IF ($FLAG[M_Test_GrdstFahren1] AND NOT $FLAG[M_Test_GrdstFahren2]) THEN
  $FLAG[M_Test_GrdstFahren2]=TRUE
  UP_Rueckzug( )
  RETURN
ENDIF
;ENDFOLD

;-------------------------------
; Place part position
;-------------------------------
TRIGGER WHEN DISTANCE=1 DELAY=-1 DO Schrittmerker_R1Place(10553,10554,FPlace_R1_L5_S2_AP,XPlace_R1_L5_S2_AP) PRIO=-1
;FOLD LIN Place_R1_L5_S2_AP Vel=0.2 m/s LPlace_R1_L5_S2_AP Tool[1]:Upper Gripper Base[1]:Rack1;%{PE}%R8.3.21,%MKUKATPBASIS,%CMOVE,%VLIN,%P 1:LIN, 2:Place_R1_L5_S2_AP, 3:, 5:0.2, 7:LPlace_R1_L5_S2_AP
$BWDSTART=FALSE
LDAT_ACT= LLPlace_R1_L5_S2_AP
FDAT_ACT= FPlace_R1_L5_S2_AP
BAS(#CP_PARAMS,0.2)
LIN XPlace_R1_L5_S2_AP
;ENDFOLD

;FOLD Test the way back home - part 2
CONTINUE
IF $FLAG[M_Test_GrdstFahren2] THEN
  $FLAG[M_Test_GrdstFahren2]=FALSE
  UP_Rueckzug( )
  RETURN
ENDIF
;ENDFOLD

;***************************************************
; Disable part lost detection
SetPartLostDetection(NO_PART)
;***************************************************

TRIGGER WHEN DISTANCE=1 DELAY=-1 DO Schrittmerker_R1Place(10554,10555,FPlace_R1_L5_S2_NP1,XPlace_R1_L5_S2_NP1) PRIO=-1
;FOLD LIN Place_R1_L5_S2_NP1 Vel=0.2 m/s LPlace_R1_L5_S2_NP1 Tool[1]:Upper Gripper Base[1]:Rack1;%{PE}%R8.3.21,%MKUKATPBASIS,%CMOVE,%VLIN,%P 1:LIN, 2:Place_R1_L5_S2_NP1, 3:C_DIS C_DIS, 5:0.2, 7:LPlace_R1_L5_S2_NP1
$BWDSTART=FALSE
LDAT_ACT= LLPlace_R1_L5_S2_NP1
FDAT_ACT= FPlace_R1_L5_S2_NP1
BAS(#CP_PARAMS,0.2)
LIN XPlace_R1_L5_S2_NP1
;ENDFOLD

;***************************************************
; Check for part present (empty gripper)
CheckPartPresent(EMPTY_GRIPPER)
;***************************************************
; set load data
SetLoadData( )
;***************************************************

TRIGGER WHEN DISTANCE=1 DELAY=-1 DO Schrittmerker_R1Place(10555,10556,FPlace_R1_L5_S2_NP2,XPlace_R1_L5_S2_NP2) PRIO=-1
;FOLD LIN Place_R1_L5_S2_NP2 CONT Vel=0.5 m/s LPlace_R1_L5_S2_NP2 Tool[1]:Upper Gripper Base[1]:Rack1;%{PE}%R8.3.21,%MKUKATPBASIS,%CMOVE,%VLIN,%P 1:LIN, 2:Place_R1_L5_S2_NP2, 3:C_DIS C_DIS, 5:0.5, 7:LPlace_R1_L5_S2_NP2
$BWDSTART=FALSE
LDAT_ACT= LLPlace_R1_L5_S2_NP2
FDAT_ACT= FPlace_R1_L5_S2_NP2
BAS(#CP_PARAMS,0.5)
LIN XPlace_R1_L5_S2_NP2 C_DIS C_DIS
;ENDFOLD
TRIGGER WHEN DISTANCE=1 DELAY=-1 DO Schrittmerker_R1Place(10556,10557,FPlace_R1_L5_S2_NP3,XPlace_R1_L5_S2_NP3) PRIO=-1
;FOLD LIN Place_R1_L5_S2_NP3 CONT Vel=0.5 m/s LPlace_R1_L5_S2_NP3 Tool[1]:Upper Gripper Base[1]:Rack1;%{PE}%R8.3.21,%MKUKATPBASIS,%CMOVE,%VLIN,%P 1:LIN, 2:Place_R1_L5_S2_NP3, 3:C_DIS C_DIS, 5:0.5, 7:LPlace_R1_L5_S2_NP3
$BWDSTART=FALSE
LDAT_ACT= LLPlace_R1_L5_S2_NP3
FDAT_ACT= FPlace_R1_L5_S2_NP3
BAS(#CP_PARAMS,0.5)
LIN XPlace_R1_L5_S2_NP3 C_DIS C_DIS
;ENDFOLD
TRIGGER WHEN DISTANCE=1 DELAY=-1 DO Schrittmerker_R1Place(10557,10558,FPlace_R1_L5_S2_NP4,XPlace_R1_L5_S2_NP4) PRIO=-1
;FOLD LIN Place_R1_L5_S2_NP4 Vel=0.5 m/s LPlace_R1_L5_S2_NP4 Tool[1]:Upper Gripper Base[1]:Rack1;%{PE}%R8.3.21,%MKUKATPBASIS,%CMOVE,%VLIN,%P 1:LIN, 2:Place_R1_L5_S2_NP4, 3:, 5:0.5, 7:LPlace_R1_L5_S2_NP4
$BWDSTART=FALSE
LDAT_ACT= LLPlace_R1_L5_S2_NP4
FDAT_ACT= FPlace_R1_L5_S2_NP4
BAS(#CP_PARAMS,0.5)
LIN XPlace_R1_L5_S2_NP4
;ENDFOLD
TRIGGER WHEN DISTANCE=1 DELAY=-1 DO Schrittmerker_R1Place(10558,10559,FPlace_R1_L5_S2_NP5,XPlace_R1_L5_S2_NP5) PRIO=-1
;FOLD PTP Place_R1_L5_S2_NP5 CONT Vel=100 % PPlace_R1_L5_S2_NP5 Tool[1]:Upper Gripper Base[0];%{PE}%R8.3.21,%MKUKATPBASIS,%CMOVE,%VPTP,%P 1:PTP, 2:Place_R1_L5_S2_NP5, 3:C_DIS, 5:100, 7:PPlace_R1_L5_S2_NP5
$BWDSTART=FALSE
PDAT_ACT= PPPlace_R1_L5_S2_NP5
FDAT_ACT= FPlace_R1_L5_S2_NP5
BAS(#PTP_PARAMS,100)
PTP XPlace_R1_L5_S2_NP5 C_DIS
;ENDFOLD
TRIGGER WHEN DISTANCE=1 DELAY=-1 DO Schrittmerker_R1Place(10559,10560,FPlace_R1_L5_S2_NP6,XPlace_R1_L5_S2_NP6) PRIO=-1
;FOLD PTP Place_R1_L5_S2_NP6 CONT Vel=100 % PPlace_R1_L5_S2_NP6 Tool[1]:Upper Gripper Base[0];%{PE}%R8.3.21,%MKUKATPBASIS,%CMOVE,%VPTP,%P 1:PTP, 2:Place_R1_L5_S2_NP6, 3:C_DIS, 5:100, 7:PPlace_R1_L5_S2_NP6
$BWDSTART=FALSE
PDAT_ACT= PPPlace_R1_L5_S2_NP6
FDAT_ACT= FPlace_R1_L5_S2_NP6
BAS(#PTP_PARAMS,100)
PTP XPlace_R1_L5_S2_NP6 C_DIS
;ENDFOLD
TRIGGER WHEN DISTANCE=1 DELAY=-1 DO Schrittmerker_R1Place(10560,10561,FPlace_R1_L5_S2_NP7,XPlace_R1_L5_S2_NP7) PRIO=-1
;FOLD PTP Place_R1_L5_S2_NP7 CONT Vel=100 % PPlace_R1_L5_S2_NP7 Tool[1]:Upper Gripper Base[0];%{PE}%R8.3.21,%MKUKATPBASIS,%CMOVE,%VPTP,%P 1:PTP, 2:Place_R1_L5_S2_NP7, 3:C_DIS, 5:100, 7:PPlace_R1_L5_S2_NP7
$BWDSTART=FALSE
PDAT_ACT= PPPlace_R1_L5_S2_NP7
FDAT_ACT= FPlace_R1_L5_S2_NP7
BAS(#PTP_PARAMS,100)
PTP XPlace_R1_L5_S2_NP7 C_DIS
;ENDFOLD
TRIGGER WHEN DISTANCE=1 DELAY=-1 DO Schrittmerker_R1Place(10561,10562,FPlace_R1_L5_S2_NP8,XPlace_R1_L5_S2_NP8) PRIO=-1
;FOLD PTP Place_R1_L5_S2_NP8 CONT Vel=100 % PPlace_R1_L5_S2_NP8 Tool[1]:Upper Gripper Base[0];%{PE}%R8.3.21,%MKUKATPBASIS,%CMOVE,%VPTP,%P 1:PTP, 2:Place_R1_L5_S2_NP8, 3:C_DIS, 5:100, 7:PPlace_R1_L5_S2_NP8
$BWDSTART=FALSE
PDAT_ACT= PPPlace_R1_L5_S2_NP8
FDAT_ACT= FPlace_R1_L5_S2_NP8
BAS(#PTP_PARAMS,100)
PTP XPlace_R1_L5_S2_NP8 C_DIS
;ENDFOLD

TRIGGER WHEN DISTANCE=1 DELAY=-1 DO Schrittmerker_R1Place(10562,10501,FHOME,$nullframe,XHOME) PRIO=-1
;FOLD PTP HOME Vel=100 % PHome;%{PE}%R8.3.21,%MKUKATPBASIS,%CMOVE,%VPTP,%P 1:PTP, 2:HOME, 3:, 5:100, 7:PHome
$BWDSTART=FALSE
PDAT_ACT= PPHome
FDAT_ACT= FHOME
BAS(#PTP_PARAMS,100)
PTP XHOME
;ENDFOLD

;***************************************************
;FOLD Final tasks.
; Robot out of area Rack 1 Level 5
RobAusStorage1_5_A71=RESET_IN_AREA
;***************************************************
; stop cyclic clearence check
$CYCFLAG[ciFreigabeSPS]=DISABLE_MONITORING
;***************************************************
; Disable collision detection
;FOLD COLLDETECT Off ;%{PE}
;FOLD Parameters ;%{h}
;Params IlfProvider=kukaroboter.basistech.inlineforms.colldetect.off; CollDetect.Command=Off
;ENDFOLD
USE_CD_PARAMS(0)
;ENDFOLD
;***************************************************
;ENDFOLD
;***************************************************

END

; ##################################################

GLOBAL DEF UP_Place_R1_L5_S3( )
;***************************************************
; Place part on:
;    Rack  1
;    Level 5
;    Shelf 3
;***************************************************
;FOLD Preconditions - Vorraussetzungen
;***************************************************
; Enable collision detection
;FOLD COLLDETECT SetLimits Axis1: 150 % Axis2: 200 % Axis3: 150 % Axis4: 200 % Axis5: 150 % Axis6: 150 % ;%{PE}
;FOLD Parameters ;%{h}
;Params IlfProvider=kukaroboter.basistech.inlineforms.colldetect.setlimits; CollDetect.Command=SetLimits; CollDetect.Axis1=150; CollDetect.Axis2=200; CollDetect.Axis3=150; CollDetect.Axis4=200; CollDetect.Axis5=150; CollDetect.Axis6=150
;ENDFOLD
SET_TQ_VALUES(150, 200, 150, 200, 150, 150)
;ENDFOLD
;***************************************************
; Check for part in gripper (tool 1).
CheckPartPresent(OCCUPIED_GRIPPER,PART_ON_TOOL_1)
;***************************************************
; Enable part lost detection for tool 1
SetPartLostDetection(PART_ON_TOOL_1)
;***************************************************
; Set load data.
SetLoadData( )
;***************************************************
; Robot has to start from home position.
IF NOT $IN_HOME THEN
  UP_HomeToHome(0)
ENDIF
;***************************************************
;ENDFOLD

TRIGGER WHEN DISTANCE=1 DELAY=-1 DO Schrittmerker_R1Place(10501,10501,FHOME,$nullframe,XHOME) PRIO=-1
;FOLD PTP HOME Vel=12 % PHome;%{PE}%R8.3.21,%MKUKATPBASIS,%CMOVE,%VPTP,%P 1:PTP, 2:HOME, 3:, 5:12, 7:PHome
$BWDSTART=FALSE
PDAT_ACT= PPHome
FDAT_ACT= FHOME
BAS(#PTP_PARAMS,12)
PTP XHOME
;ENDFOLD

;***************************************************
;FOLD Area clearence handshake.
IF NOT $FLAG[M_Inbetriebnahme] THEN
  ;-------------------------------------------------
  ; Request area clearence.
  AnfStoer_Store1_5_A103=SET_REQUEST
  ;-------------------------------------------------
  ; Wait for area clearence from PLC.
  WAIT_FOR_INPUT("Frg_Storage1_5_E71",TRUE)
  ;-------------------------------------------------
  ; Reset area clearence request.
  AnfStoer_Store1_5_A103=RESET_REQUEST
  ;-------------------------------------------------
  ; start cyclic clearence check
  $CYCFLAG[ciFreigabeSPS]=Frg_Storage1_5_E71
  ;-------------------------------------------------
ENDIF
;***************************************************
; set "robot in area"
RobAusStorage1_5_A71=SET_IN_AREA
;ENDFOLD
;***************************************************

;***************************************************
;FOLD Check for Teachmode
IF $FLAG[M_Teachen] THEN
  WAIT FOR $T1
ENDIF
;ENDFOLD
;***************************************************

; move to the rack
TRIGGER WHEN DISTANCE=1 DELAY=-1 DO Schrittmerker_R1Place(10570,10501,FPlace_R1_L5_S3_VP1,XPlace_R1_L5_S3_VP1) PRIO=-1
;FOLD PTP Place_R1_L5_S3_VP1 CONT Vel=12 % PPlace_R1_L5_S3_VP1 Tool[1]:Upper Gripper Base[0];%{PE}%R8.3.21,%MKUKATPBASIS,%CMOVE,%VPTP,%P 1:PTP, 2:Place_R1_L5_S3_VP1, 3:C_DIS, 5:12, 7:PPlace_R1_L5_S3_VP1
$BWDSTART=FALSE
PDAT_ACT= PPPlace_R1_L5_S3_VP1
FDAT_ACT= FPlace_R1_L5_S3_VP1
BAS(#PTP_PARAMS,12)
PTP XPlace_R1_L5_S3_VP1 C_DIS
;ENDFOLD
TRIGGER WHEN DISTANCE=1 DELAY=-1 DO Schrittmerker_R1Place(10571,10570,FPlace_R1_L5_S3_VP2,XPlace_R1_L5_S3_VP2) PRIO=-1
;FOLD PTP Place_R1_L5_S3_VP2 CONT Vel=12 % PPlace_R1_L5_S3_VP2 Tool[1]:Upper Gripper Base[0];%{PE}%R8.3.21,%MKUKATPBASIS,%CMOVE,%VPTP,%P 1:PTP, 2:Place_R1_L5_S3_VP2, 3:C_DIS, 5:12, 7:PPlace_R1_L5_S3_VP2
$BWDSTART=FALSE
PDAT_ACT= PPPlace_R1_L5_S3_VP2
FDAT_ACT= FPlace_R1_L5_S3_VP2
BAS(#PTP_PARAMS,12)
PTP XPlace_R1_L5_S3_VP2 C_DIS
;ENDFOLD
TRIGGER WHEN DISTANCE=1 DELAY=-1 DO Schrittmerker_R1Place(10572,10571,FPlace_R1_L5_S3_VP3,XPlace_R1_L5_S3_VP3) PRIO=-1
;FOLD PTP Place_R1_L5_S3_VP3 CONT Vel=12 % PPlace_R1_L5_S3_VP3 Tool[1]:Upper Gripper Base[0];%{PE}%R8.3.21,%MKUKATPBASIS,%CMOVE,%VPTP,%P 1:PTP, 2:Place_R1_L5_S3_VP3, 3:C_DIS, 5:12, 7:PPlace_R1_L5_S3_VP3
$BWDSTART=FALSE
PDAT_ACT= PPPlace_R1_L5_S3_VP3
FDAT_ACT= FPlace_R1_L5_S3_VP3
BAS(#PTP_PARAMS,12)
PTP XPlace_R1_L5_S3_VP3 C_DIS
;ENDFOLD

TRIGGER WHEN DISTANCE=1 DELAY=-1 DO Schrittmerker_R1Place(10573,10572,FPlace_R1_L5_S3_Check,XPlace_R1_L5_S3_Check) PRIO=-1
;FOLD PTP Place_R1_L5_S3_Check Vel=12 % PPlace_R1_L5_S3_Check Tool[1]:Upper Gripper Base[1]:Rack1;%{PE}%R8.3.21,%MKUKATPBASIS,%CMOVE,%VPTP,%P 1:PTP, 2:Place_R1_L5_S3_Check, 3:, 5:12, 7:PPlace_R1_L5_S3_Check
$BWDSTART=FALSE
PDAT_ACT= PPPlace_R1_L5_S3_Check
FDAT_ACT= FPlace_R1_L5_S3_Check
BAS(#PTP_PARAMS,12)
PTP XPlace_R1_L5_S3_Check
;ENDFOLD

;***************************************************
;FOLD Pruefe Platz frei
IF (DetectPart(CHECK_SHELF,PLACE)==OCCUPIED) THEN
  UP_Rueckzug_R1Place( )
  RETURN
ENDIF
;ENDFOLD
;***************************************************

TRIGGER WHEN DISTANCE=1 DELAY=-1 DO Schrittmerker_R1Place(10574,10573,FPlace_R1_L5_S3_VP4,XPlace_R1_L5_S3_VP4) PRIO=-1
;FOLD LIN Place_R1_L5_S3_VP4 CONT Vel=0.5 m/s LPlace_R1_L5_S3_VP4 Tool[1]:Upper Gripper Base[1]:Rack1;%{PE}%R8.3.21,%MKUKATPBASIS,%CMOVE,%VLIN,%P 1:LIN, 2:Place_R1_L5_S3_VP4, 3:C_DIS C_DIS, 5:0.5, 7:LPlace_R1_L5_S3_VP4
$BWDSTART=FALSE
LDAT_ACT= LLPlace_R1_L5_S3_VP4
FDAT_ACT= FPlace_R1_L5_S3_VP4
BAS(#CP_PARAMS,0.5)
LIN XPlace_R1_L5_S3_VP4 C_DIS C_DIS
;ENDFOLD
TRIGGER WHEN DISTANCE=1 DELAY=-1 DO Schrittmerker_R1Place(10575,10574,FPlace_R1_L5_S3_VP5,XPlace_R1_L5_S3_VP5) PRIO=-1
;FOLD LIN Place_R1_L5_S3_VP5 CONT Vel=0.5 m/s LPlace_R1_L5_S3_VP5 Tool[1]:Upper Gripper Base[1]:Rack1;%{PE}%R8.3.21,%MKUKATPBASIS,%CMOVE,%VLIN,%P 1:LIN, 2:Place_R1_L5_S3_VP5, 3:C_DIS C_DIS, 5:0.5, 7:LPlace_R1_L5_S3_VP5
$BWDSTART=FALSE
LDAT_ACT= LLPlace_R1_L5_S3_VP5
FDAT_ACT= FPlace_R1_L5_S3_VP5
BAS(#CP_PARAMS,0.5)
LIN XPlace_R1_L5_S3_VP5 C_DIS C_DIS
;ENDFOLD
TRIGGER WHEN DISTANCE=1 DELAY=-1 DO Schrittmerker_R1Place(10576,10575,FPlace_R1_L5_S3_VP6,XPlace_R1_L5_S3_VP6) PRIO=-1
;FOLD LIN Place_R1_L5_S3_VP6 CONT Vel=0.5 m/s LPlace_R1_L5_S3_VP6 Tool[1]:Upper Gripper Base[1]:Rack1;%{PE}%R8.3.21,%MKUKATPBASIS,%CMOVE,%VLIN,%P 1:LIN, 2:Place_R1_L5_S3_VP6, 3:C_DIS C_DIS, 5:0.5, 7:LPlace_R1_L5_S3_VP6
$BWDSTART=FALSE
LDAT_ACT= LLPlace_R1_L5_S3_VP6
FDAT_ACT= FPlace_R1_L5_S3_VP6
BAS(#CP_PARAMS,0.5)
LIN XPlace_R1_L5_S3_VP6 C_DIS C_DIS
;ENDFOLD

;FOLD Test the way back home - part 1
CONTINUE
IF ($FLAG[M_Test_GrdstFahren1] AND NOT $FLAG[M_Test_GrdstFahren2]) THEN
  $FLAG[M_Test_GrdstFahren2]=TRUE
  UP_Rueckzug( )
  RETURN
ENDIF
;ENDFOLD

;-------------------------------
; Place part position
;-------------------------------
TRIGGER WHEN DISTANCE=1 DELAY=-1 DO Schrittmerker_R1Place(10577,10578,FPlace_R1_L5_S3_AP,XPlace_R1_L5_S3_AP) PRIO=-1
;FOLD LIN Place_R1_L5_S3_AP Vel=0.2 m/s LPlace_R1_L5_S3_AP Tool[1]:Upper Gripper Base[1]:Rack1;%{PE}%R8.3.21,%MKUKATPBASIS,%CMOVE,%VLIN,%P 1:LIN, 2:Place_R1_L5_S3_AP, 3:, 5:0.2, 7:LPlace_R1_L5_S3_AP
$BWDSTART=FALSE
LDAT_ACT= LLPlace_R1_L5_S3_AP
FDAT_ACT= FPlace_R1_L5_S3_AP
BAS(#CP_PARAMS,0.2)
LIN XPlace_R1_L5_S3_AP
;ENDFOLD

;FOLD Test the way back home - part 2
CONTINUE
IF $FLAG[M_Test_GrdstFahren2] THEN
  $FLAG[M_Test_GrdstFahren2]=FALSE
  UP_Rueckzug( )
  RETURN
ENDIF
;ENDFOLD

;***************************************************
; Disable part lost detection
SetPartLostDetection(NO_PART)
;***************************************************

TRIGGER WHEN DISTANCE=1 DELAY=-1 DO Schrittmerker_R1Place(10578,10579,FPlace_R1_L5_S3_NP1,XPlace_R1_L5_S3_NP1) PRIO=-1
;FOLD LIN Place_R1_L5_S3_NP1 Vel=0.2 m/s LPlace_R1_L5_S3_NP1 Tool[1]:Upper Gripper Base[1]:Rack1;%{PE}%R8.3.21,%MKUKATPBASIS,%CMOVE,%VLIN,%P 1:LIN, 2:Place_R1_L5_S3_NP1, 3:C_DIS C_DIS, 5:0.2, 7:LPlace_R1_L5_S3_NP1
$BWDSTART=FALSE
LDAT_ACT= LLPlace_R1_L5_S3_NP1
FDAT_ACT= FPlace_R1_L5_S3_NP1
BAS(#CP_PARAMS,0.2)
LIN XPlace_R1_L5_S3_NP1
;ENDFOLD

;***************************************************
; Check for part present (empty gripper)
CheckPartPresent(EMPTY_GRIPPER)
;***************************************************
; set load data
SetLoadData( )
;***************************************************

TRIGGER WHEN DISTANCE=1 DELAY=-1 DO Schrittmerker_R1Place(10579,10580,FPlace_R1_L5_S3_NP2,XPlace_R1_L5_S3_NP2) PRIO=-1
;FOLD LIN Place_R1_L5_S3_NP2 Vel=0.5 m/s LPlace_R1_L5_S3_NP2 Tool[1]:Upper Gripper Base[1]:Rack 1 ;%{PE}
$BWDSTART = FALSE
LDAT_ACT = LLPlace_R1_L5_S3_NP2
FDAT_ACT = FPlace_R1_L5_S3_NP2
BAS(#CP_PARAMS, 0.5)
LIN XPlace_R1_L5_S3_NP2
;ENDFOLD
TRIGGER WHEN DISTANCE=1 DELAY=-1 DO Schrittmerker_R1Place(10580,10581,FPlace_R1_L5_S3_NP3,XPlace_R1_L5_S3_NP3) PRIO=-1
;FOLD PTP Place_R1_L5_S3_NP3 CONT Vel=100 % PPlace_R1_L5_S3_NP3 Tool[1]:Upper Gripper Base[1]:Rack1;%{PE}%R8.3.21,%MKUKATPBASIS,%CMOVE,%VPTP,%P 1:PTP, 2:Place_R1_L5_S3_NP3, 3:C_DIS, 5:100, 7:PPlace_R1_L5_S3_NP3
$BWDSTART=FALSE
PDAT_ACT= PPPlace_R1_L5_S3_NP3
FDAT_ACT= FPlace_R1_L5_S3_NP3
BAS(#PTP_PARAMS,100)
PTP XPlace_R1_L5_S3_NP3 C_DIS
;ENDFOLD
TRIGGER WHEN DISTANCE=1 DELAY=-1 DO Schrittmerker_R1Place(10581,10582,FPlace_R1_L5_S3_NP4,XPlace_R1_L5_S3_NP4) PRIO=-1
;FOLD PTP Place_R1_L5_S3_NP4 CONT Vel=100 % PPlace_R1_L5_S3_NP4 Tool[1]:Upper Gripper Base[0];%{PE}%R8.3.21,%MKUKATPBASIS,%CMOVE,%VPTP,%P 1:PTP, 2:Place_R1_L5_S3_NP4, 3:C_DIS, 5:100, 7:PPlace_R1_L5_S3_NP4
$BWDSTART=FALSE
PDAT_ACT= PPPlace_R1_L5_S3_NP4
FDAT_ACT= FPlace_R1_L5_S3_NP4
BAS(#PTP_PARAMS,100)
PTP XPlace_R1_L5_S3_NP4 C_DIS
;ENDFOLD
TRIGGER WHEN DISTANCE=1 DELAY=-1 DO Schrittmerker_R1Place(10582,10583,FPlace_R1_L5_S3_NP5,XPlace_R1_L5_S3_NP5) PRIO=-1
;FOLD PTP Place_R1_L5_S3_NP5 CONT Vel=100 % PPlace_R1_L5_S3_NP5 Tool[1]:Upper Gripper Base[0];%{PE}%R8.3.21,%MKUKATPBASIS,%CMOVE,%VPTP,%P 1:PTP, 2:Place_R1_L5_S3_NP5, 3:C_DIS, 5:100, 7:PPlace_R1_L5_S3_NP5
$BWDSTART=FALSE
PDAT_ACT= PPPlace_R1_L5_S3_NP5
FDAT_ACT= FPlace_R1_L5_S3_NP5
BAS(#PTP_PARAMS,100)
PTP XPlace_R1_L5_S3_NP5 C_DIS
;ENDFOLD

TRIGGER WHEN DISTANCE=1 DELAY=-1 DO Schrittmerker_R1Place(10583,10501,FHOME,$nullframe,XHOME) PRIO=-1
;FOLD PTP HOME Vel=100 % PHome;%{PE}%R8.3.21,%MKUKATPBASIS,%CMOVE,%VPTP,%P 1:PTP, 2:HOME, 3:, 5:100, 7:PHome
$BWDSTART=FALSE
PDAT_ACT= PPHome
FDAT_ACT= FHOME
BAS(#PTP_PARAMS,100)
PTP XHOME
;ENDFOLD

;***************************************************
;FOLD Final tasks.
; Robot out of area Rack 1 Level 5
RobAusStorage1_5_A71=RESET_IN_AREA
;***************************************************
; stop cyclic clearence check
$CYCFLAG[ciFreigabeSPS]=DISABLE_MONITORING
;***************************************************
; Disable collision detection
;FOLD COLLDETECT Off ;%{PE}
;FOLD Parameters ;%{h}
;Params IlfProvider=kukaroboter.basistech.inlineforms.colldetect.off; CollDetect.Command=Off
;ENDFOLD
USE_CD_PARAMS(0)
;ENDFOLD
;***************************************************
;ENDFOLD
;***************************************************

END

; ##################################################

GLOBAL DEF UP_Place_R1_L5_S4( )
;***************************************************
; Place part on:
;    Rack  1
;    Level 5
;    Shelf 4
;***************************************************
;FOLD Preconditions - Vorraussetzungen
;***************************************************
; Enable collision detection
;FOLD COLLDETECT SetLimits Axis1: 150 % Axis2: 200 % Axis3: 150 % Axis4: 200 % Axis5: 150 % Axis6: 150 % ;%{PE}
;FOLD Parameters ;%{h}
;Params IlfProvider=kukaroboter.basistech.inlineforms.colldetect.setlimits; CollDetect.Command=SetLimits; CollDetect.Axis1=150; CollDetect.Axis2=200; CollDetect.Axis3=150; CollDetect.Axis4=200; CollDetect.Axis5=150; CollDetect.Axis6=150
;ENDFOLD
SET_TQ_VALUES(150, 200, 150, 200, 150, 150)
;ENDFOLD
;***************************************************
; Check for part in gripper (tool 1).
CheckPartPresent(OCCUPIED_GRIPPER,PART_ON_TOOL_1)
;***************************************************
; Enable part lost detection for tool 1
SetPartLostDetection(PART_ON_TOOL_1)
;***************************************************
; Set load data.
SetLoadData( )
;***************************************************
; Robot has to start from home position.
IF NOT $IN_HOME THEN
  UP_HomeToHome(0)
ENDIF
;***************************************************
;ENDFOLD

TRIGGER WHEN DISTANCE=1 DELAY=-1 DO Schrittmerker_R1Place(10501,10501,FHOME,$nullframe,XHOME) PRIO=-1
;FOLD PTP HOME Vel=12 % PHome;%{PE}%R8.3.21,%MKUKATPBASIS,%CMOVE,%VPTP,%P 1:PTP, 2:HOME, 3:, 5:12, 7:PHome
$BWDSTART=FALSE
PDAT_ACT= PPHome
FDAT_ACT= FHOME
BAS(#PTP_PARAMS,12)
PTP XHOME
;ENDFOLD

;***************************************************
;FOLD Area clearence handshake.
IF NOT $FLAG[M_Inbetriebnahme] THEN
  ;-------------------------------------------------
  ; Request area clearence.
  AnfStoer_Store1_5_A103=SET_REQUEST
  ;-------------------------------------------------
  ; Wait for area clearence from PLC.
  WAIT_FOR_INPUT("Frg_Storage1_5_E71",TRUE)
  ;-------------------------------------------------
  ; Reset area clearence request.
  AnfStoer_Store1_5_A103=RESET_REQUEST
  ;-------------------------------------------------
  ; start cyclic clearence check
  $CYCFLAG[ciFreigabeSPS]=Frg_Storage1_5_E71
  ;-------------------------------------------------
ENDIF
;***************************************************
; set "robot in area"
RobAusStorage1_5_A71=SET_IN_AREA
;ENDFOLD
;***************************************************

;***************************************************
;FOLD Check for Teachmode
IF $FLAG[M_Teachen] THEN
  WAIT FOR $T1
ENDIF
;ENDFOLD
;***************************************************

; move to the rack
TRIGGER WHEN DISTANCE=1 DELAY=-1 DO Schrittmerker_R1Place(10590,10501,FPlace_R1_L5_S4_VP1,XPlace_R1_L5_S4_VP1) PRIO=-1
;FOLD PTP Place_R1_L5_S4_VP1 CONT Vel=12 % PPlace_R1_L5_S4_VP1 Tool[1]:Upper Gripper Base[0];%{PE}%R8.3.21,%MKUKATPBASIS,%CMOVE,%VPTP,%P 1:PTP, 2:Place_R1_L5_S4_VP1, 3:C_DIS, 5:12, 7:PPlace_R1_L5_S4_VP1
$BWDSTART=FALSE
PDAT_ACT= PPPlace_R1_L5_S4_VP1
FDAT_ACT= FPlace_R1_L5_S4_VP1
BAS(#PTP_PARAMS,12)
PTP XPlace_R1_L5_S4_VP1 C_DIS
;ENDFOLD
TRIGGER WHEN DISTANCE=1 DELAY=-1 DO Schrittmerker_R1Place(10591,10590,FPlace_R1_L5_S4_VP2,XPlace_R1_L5_S4_VP2) PRIO=-1
;FOLD PTP Place_R1_L5_S4_VP2 CONT Vel=12 % PPlace_R1_L5_S4_VP2 Tool[1]:Upper Gripper Base[0];%{PE}%R8.3.21,%MKUKATPBASIS,%CMOVE,%VPTP,%P 1:PTP, 2:Place_R1_L5_S4_VP2, 3:C_DIS, 5:12, 7:PPlace_R1_L5_S4_VP2
$BWDSTART=FALSE
PDAT_ACT= PPPlace_R1_L5_S4_VP2
FDAT_ACT= FPlace_R1_L5_S4_VP2
BAS(#PTP_PARAMS,12)
PTP XPlace_R1_L5_S4_VP2 C_DIS
;ENDFOLD
TRIGGER WHEN DISTANCE=1 DELAY=-1 DO Schrittmerker_R1Place(10592,10591,FPlace_R1_L5_S4_VP3,XPlace_R1_L5_S4_VP3) PRIO=-1
;FOLD PTP Place_R1_L5_S4_VP3 CONT Vel=12 % PPlace_R1_L5_S4_VP3 Tool[1]:Upper Gripper Base[0];%{PE}%R8.3.21,%MKUKATPBASIS,%CMOVE,%VPTP,%P 1:PTP, 2:Place_R1_L5_S4_VP3, 3:C_DIS, 5:12, 7:PPlace_R1_L5_S4_VP3
$BWDSTART=FALSE
PDAT_ACT= PPPlace_R1_L5_S4_VP3
FDAT_ACT= FPlace_R1_L5_S4_VP3
BAS(#PTP_PARAMS,12)
PTP XPlace_R1_L5_S4_VP3 C_DIS
;ENDFOLD
TRIGGER WHEN DISTANCE=1 DELAY=-1 DO Schrittmerker_R1Place(10593,10592,FPlace_R1_L5_S4_VP4,XPlace_R1_L5_S4_VP4) PRIO=-1
;FOLD PTP Place_R1_L5_S4_VP4 CONT Vel=12 % PPlace_R1_L5_S4_VP4 Tool[1]:Upper Gripper Base[1]:Rack1;%{PE}%R8.3.21,%MKUKATPBASIS,%CMOVE,%VPTP,%P 1:PTP, 2:Place_R1_L5_S4_VP4, 3:C_DIS, 5:12, 7:PPlace_R1_L5_S4_VP4
$BWDSTART=FALSE
PDAT_ACT= PPPlace_R1_L5_S4_VP4
FDAT_ACT= FPlace_R1_L5_S4_VP4
BAS(#PTP_PARAMS,12)
PTP XPlace_R1_L5_S4_VP4 C_DIS
;ENDFOLD

TRIGGER WHEN DISTANCE=1 DELAY=-1 DO Schrittmerker_R1Place(10594,10593,FPlace_R1_L5_S4_Check,XPlace_R1_L5_S4_Check) PRIO=-1
;FOLD PTP Place_R1_L5_S4_Check Vel=12 % PPlace_R1_L5_S4_Check Tool[1]:Upper Gripper Base[1]:Rack1;%{PE}%R8.3.21,%MKUKATPBASIS,%CMOVE,%VPTP,%P 1:PTP, 2:Place_R1_L5_S4_Check, 3:, 5:12, 7:PPlace_R1_L5_S4_Check
$BWDSTART=FALSE
PDAT_ACT= PPPlace_R1_L5_S4_Check
FDAT_ACT= FPlace_R1_L5_S4_Check
BAS(#PTP_PARAMS,12)
PTP XPlace_R1_L5_S4_Check
;ENDFOLD

;***************************************************
;FOLD Pruefe Platz frei
IF (DetectPart(CHECK_SHELF,PLACE)==OCCUPIED) THEN
  UP_Rueckzug_R1Place( )
  RETURN
ENDIF
;ENDFOLD
;***************************************************

TRIGGER WHEN DISTANCE=1 DELAY=-1 DO Schrittmerker_R1Place(10595,10594,FPlace_R1_L5_S4_VP5,XPlace_R1_L5_S4_VP5) PRIO=-1
;FOLD LIN Place_R1_L5_S4_VP5 CONT Vel=0.5 m/s LPlace_R1_L5_S4_VP5 Tool[1]:Upper Gripper Base[1]:Rack1;%{PE}%R8.3.21,%MKUKATPBASIS,%CMOVE,%VLIN,%P 1:LIN, 2:Place_R1_L5_S4_VP5, 3:C_DIS C_DIS, 5:0.5, 7:LPlace_R1_L5_S4_VP5
$BWDSTART=FALSE
LDAT_ACT= LLPlace_R1_L5_S4_VP5
FDAT_ACT= FPlace_R1_L5_S4_VP5
BAS(#CP_PARAMS,0.5)
LIN XPlace_R1_L5_S4_VP5 C_DIS C_DIS
;ENDFOLD

;***************************************************
;FOLD Test the way back home - part 1
CONTINUE
IF ($FLAG[M_Test_GrdstFahren1] AND NOT $FLAG[M_Test_GrdstFahren2]) THEN
  $FLAG[M_Test_GrdstFahren2]=TRUE
  UP_Rueckzug( )
  RETURN
ENDIF
;ENDFOLD
;***************************************************

;-------------------------------
; Place part position
;-------------------------------
TRIGGER WHEN DISTANCE=1 DELAY=-1 DO Schrittmerker_R1Place(10596,10597,FPlace_R1_L5_S4_AP,XPlace_R1_L5_S4_AP) PRIO=-1
;FOLD LIN Place_R1_L5_S4_AP Vel=0.2 m/s LPlace_R1_L5_S4_AP Tool[1]:Upper Gripper Base[1]:Rack1;%{PE}%R8.3.21,%MKUKATPBASIS,%CMOVE,%VLIN,%P 1:LIN, 2:Place_R1_L5_S4_AP, 3:, 5:0.2, 7:LPlace_R1_L5_S4_AP
$BWDSTART=FALSE
LDAT_ACT= LLPlace_R1_L5_S4_AP
FDAT_ACT= FPlace_R1_L5_S4_AP
BAS(#CP_PARAMS,0.2)
LIN XPlace_R1_L5_S4_AP
;ENDFOLD

;FOLD Test the way back home - part 2
CONTINUE
IF $FLAG[M_Test_GrdstFahren2] THEN
  $FLAG[M_Test_GrdstFahren2]=FALSE
  UP_Rueckzug( )
  RETURN
ENDIF
;ENDFOLD

;***************************************************
; Disable part lost detection
SetPartLostDetection(NO_PART)
;***************************************************

TRIGGER WHEN DISTANCE=1 DELAY=-1 DO Schrittmerker_R1Place(10597,10598,FPlace_R1_L5_S4_NP1,XPlace_R1_L5_S4_NP1) PRIO=-1
;FOLD LIN Place_R1_L5_S4_NP1 Vel=0.2 m/s LPlace_R1_L5_S4_NP1 Tool[1]:Upper Gripper Base[1]:Rack1;%{PE}%R8.3.21,%MKUKATPBASIS,%CMOVE,%VLIN,%P 1:LIN, 2:Place_R1_L5_S4_NP1, 3:C_DIS C_DIS, 5:0.2, 7:LPlace_R1_L5_S4_NP1
$BWDSTART=FALSE
LDAT_ACT= LLPlace_R1_L5_S4_NP1
FDAT_ACT= FPlace_R1_L5_S4_NP1
BAS(#CP_PARAMS,0.2)
LIN XPlace_R1_L5_S4_NP1
;ENDFOLD

;***************************************************
; Check for part present (empty gripper)
CheckPartPresent(EMPTY_GRIPPER)
;***************************************************
; set load data
SetLoadData( )
;***************************************************

TRIGGER WHEN DISTANCE=1 DELAY=-1 DO Schrittmerker_R1Place(10598,10599,FPlace_R1_L5_S4_NP2,XPlace_R1_L5_S4_NP2) PRIO=-1
;FOLD LIN Place_R1_L5_S4_NP2 Vel=0.5 m/s LPlace_R1_L5_S4_NP2 Tool[1]:Upper Gripper Base[1]:Rack1;%{PE}%R8.3.21,%MKUKATPBASIS,%CMOVE,%VLIN,%P 1:LIN, 2:Place_R1_L5_S4_NP2, 3:, 5:0.5, 7:LPlace_R1_L5_S4_NP2
$BWDSTART=FALSE
LDAT_ACT= LLPlace_R1_L5_S4_NP2
FDAT_ACT= FPlace_R1_L5_S4_NP2
BAS(#CP_PARAMS,0.5)
LIN XPlace_R1_L5_S4_NP2
;ENDFOLD
TRIGGER WHEN DISTANCE=1 DELAY=-1 DO Schrittmerker_R1Place(10599,10600,FPlace_R1_L5_S4_NP3,XPlace_R1_L5_S4_NP3) PRIO=-1
;FOLD PTP Place_R1_L5_S4_NP3 CONT Vel=100 % PPlace_R1_L5_S4_NP3 Tool[1]:Upper Gripper Base[1]:Rack1;%{PE}%R8.3.21,%MKUKATPBASIS,%CMOVE,%VPTP,%P 1:PTP, 2:Place_R1_L5_S4_NP3, 3:C_DIS, 5:100, 7:PPlace_R1_L5_S4_NP3
$BWDSTART=FALSE
PDAT_ACT= PPPlace_R1_L5_S4_NP3
FDAT_ACT= FPlace_R1_L5_S4_NP3
BAS(#PTP_PARAMS,100)
PTP XPlace_R1_L5_S4_NP3 C_DIS
;ENDFOLD
TRIGGER WHEN DISTANCE=1 DELAY=-1 DO Schrittmerker_R1Place(10600,10601,FPlace_R1_L5_S4_NP4,XPlace_R1_L5_S4_NP4) PRIO=-1
;FOLD PTP Place_R1_L5_S4_NP4 CONT Vel=100 % PPlace_R1_L5_S4_NP4 Tool[1]:Upper Gripper Base[0];%{PE}%R8.3.21,%MKUKATPBASIS,%CMOVE,%VPTP,%P 1:PTP, 2:Place_R1_L5_S4_NP4, 3:C_DIS, 5:100, 7:PPlace_R1_L5_S4_NP4
$BWDSTART=FALSE
PDAT_ACT= PPPlace_R1_L5_S4_NP4
FDAT_ACT= FPlace_R1_L5_S4_NP4
BAS(#PTP_PARAMS,100)
PTP XPlace_R1_L5_S4_NP4 C_DIS
;ENDFOLD
TRIGGER WHEN DISTANCE=1 DELAY=-1 DO Schrittmerker_R1Place(10601,10602,FPlace_R1_L5_S4_NP5,XPlace_R1_L5_S4_NP5) PRIO=-1
;FOLD PTP Place_R1_L5_S4_NP5 CONT Vel=100 % PPlace_R1_L5_S4_NP5 Tool[1]:Upper Gripper Base[0];%{PE}%R8.3.21,%MKUKATPBASIS,%CMOVE,%VPTP,%P 1:PTP, 2:Place_R1_L5_S4_NP5, 3:C_DIS, 5:100, 7:PPlace_R1_L5_S4_NP5
$BWDSTART=FALSE
PDAT_ACT= PPPlace_R1_L5_S4_NP5
FDAT_ACT= FPlace_R1_L5_S4_NP5
BAS(#PTP_PARAMS,100)
PTP XPlace_R1_L5_S4_NP5 C_DIS
;ENDFOLD

TRIGGER WHEN DISTANCE=1 DELAY=-1 DO Schrittmerker_R1Place(10602,10501,FHOME,$nullframe,XHOME) PRIO=-1
;FOLD PTP HOME Vel=100 % PHome;%{PE}%R8.3.21,%MKUKATPBASIS,%CMOVE,%VPTP,%P 1:PTP, 2:HOME, 3:, 5:100, 7:PHome
$BWDSTART=FALSE
PDAT_ACT= PPHome
FDAT_ACT= FHOME
BAS(#PTP_PARAMS,100)
PTP XHOME
;ENDFOLD

;***************************************************
;FOLD Final tasks.
; Robot out of area Rack 1 Level 5
RobAusStorage1_5_A71=RESET_IN_AREA
;***************************************************
; stop cyclic clearence check
$CYCFLAG[ciFreigabeSPS]=DISABLE_MONITORING
;***************************************************
; Disable collision detection
;FOLD COLLDETECT Off ;%{PE}
;FOLD Parameters ;%{h}
;Params IlfProvider=kukaroboter.basistech.inlineforms.colldetect.off; CollDetect.Command=Off
;ENDFOLD
USE_CD_PARAMS(0)
;ENDFOLD
;***************************************************
;ENDFOLD
;***************************************************

END

; ##################################################

GLOBAL DEF UP_Place_R1_L6_S1( )
;***************************************************
; Place part on:
;    Rack  1
;    Level 6
;    Shelf 1
;  RBG Kollision beachten!
;***************************************************
;FOLD Preconditions - Vorraussetzungen
;***************************************************
; Enable collision detection
;FOLD COLLDETECT SetLimits Axis1: 150 % Axis2: 200 % Axis3: 150 % Axis4: 200 % Axis5: 150 % Axis6: 150 % ;%{PE}
;FOLD Parameters ;%{h}
;Params IlfProvider=kukaroboter.basistech.inlineforms.colldetect.setlimits; CollDetect.Command=SetLimits; CollDetect.Axis1=150; CollDetect.Axis2=200; CollDetect.Axis3=150; CollDetect.Axis4=200; CollDetect.Axis5=150; CollDetect.Axis6=150
;ENDFOLD
SET_TQ_VALUES(150, 200, 150, 200, 150, 150)
;ENDFOLD
;***************************************************
; Check for part in gripper (tool 1).
CheckPartPresent(OCCUPIED_GRIPPER,PART_ON_TOOL_1)
;***************************************************
; Enable part lost detection for tool 1
SetPartLostDetection(PART_ON_TOOL_1)
;***************************************************
; Set load data.
SetLoadData( )
;***************************************************
; Robot has to start from home position.
IF NOT $IN_HOME THEN
  UP_HomeToHome(0)
ENDIF
;***************************************************
;ENDFOLD

TRIGGER WHEN DISTANCE=1 DELAY=-1 DO Schrittmerker_R1Place(10501,10501,FHOME,$nullframe,XHOME) PRIO=-1
;FOLD PTP HOME Vel=12 % PHome;%{PE}%R8.3.21,%MKUKATPBASIS,%CMOVE,%VPTP,%P 1:PTP, 2:HOME, 3:, 5:12, 7:PHome
$BWDSTART=FALSE
PDAT_ACT= PPHome
FDAT_ACT= FHOME
BAS(#PTP_PARAMS,12)
PTP XHOME
;ENDFOLD

;***************************************************
;FOLD Area clearence handshake.
IF NOT $FLAG[M_Inbetriebnahme] THEN
  ;-------------------------------------------------
  ; Request area clearence.
  AnfStoer_Store1_6_A104=SET_REQUEST
  ;-------------------------------------------------
  ; Wait for area clearence from PLC.
  WAIT_FOR_INPUT("Frg_Storage1_6_E72",TRUE)
  ;-------------------------------------------------
  ; Reset area clearence request.
  AnfStoer_Store1_6_A104=RESET_REQUEST
  ;-------------------------------------------------
  ; start cyclic clearence check
  $CYCFLAG[ciFreigabeSPS]=Frg_Storage1_6_E72
  ;-------------------------------------------------
ENDIF
;***************************************************
; set "robot in area"
RobAusStorage1_6_A72=SET_IN_AREA
;ENDFOLD
;***************************************************

;***************************************************
;FOLD Check for Teachmode
IF $FLAG[M_Teachen] THEN
  WAIT FOR $T1
ENDIF
;ENDFOLD
;***************************************************

; move to the rack
TRIGGER WHEN DISTANCE=1 DELAY=-1 DO Schrittmerker_R1Place(10610,10501,FPlace_R1_L6_S1_VP1,XPlace_R1_L6_S1_VP1) PRIO=-1
;FOLD PTP Place_R1_L6_S1_VP1 CONT Vel=12 % PPlace_R1_L6_S1_VP1 Tool[1]:Upper Gripper Base[0];%{PE}%R8.3.21,%MKUKATPBASIS,%CMOVE,%VPTP,%P 1:PTP, 2:Place_R1_L6_S1_VP1, 3:C_DIS, 5:12, 7:PPlace_R1_L6_S1_VP1
$BWDSTART=FALSE
PDAT_ACT= PPPlace_R1_L6_S1_VP1
FDAT_ACT= FPlace_R1_L6_S1_VP1
BAS(#PTP_PARAMS,12)
PTP XPlace_R1_L6_S1_VP1 C_DIS
;ENDFOLD
TRIGGER WHEN DISTANCE=1 DELAY=-1 DO Schrittmerker_R1Place(10611,10610,FPlace_R1_L6_S1_VP2,XPlace_R1_L6_S1_VP2) PRIO=-1
;FOLD PTP Place_R1_L6_S1_VP2 CONT Vel=12 % PPlace_R1_L6_S1_VP2 Tool[1]:Upper Gripper Base[0];%{PE}%R8.3.21,%MKUKATPBASIS,%CMOVE,%VPTP,%P 1:PTP, 2:Place_R1_L6_S1_VP2, 3:C_DIS, 5:12, 7:PPlace_R1_L6_S1_VP2
$BWDSTART=FALSE
PDAT_ACT= PPPlace_R1_L6_S1_VP2
FDAT_ACT= FPlace_R1_L6_S1_VP2
BAS(#PTP_PARAMS,12)
PTP XPlace_R1_L6_S1_VP2 C_DIS
;ENDFOLD
TRIGGER WHEN DISTANCE=1 DELAY=-1 DO Schrittmerker_R1Place(10612,10611,FPlace_R1_L6_S1_VP3,XPlace_R1_L6_S1_VP3) PRIO=-1
;FOLD PTP Place_R1_L6_S1_VP3 CONT Vel=12 % PPlace_R1_L6_S1_VP3 Tool[1]:Upper Gripper Base[0];%{PE}%R8.3.21,%MKUKATPBASIS,%CMOVE,%VPTP,%P 1:PTP, 2:Place_R1_L6_S1_VP3, 3:C_DIS, 5:12, 7:PPlace_R1_L6_S1_VP3
$BWDSTART=FALSE
PDAT_ACT= PPPlace_R1_L6_S1_VP3
FDAT_ACT= FPlace_R1_L6_S1_VP3
BAS(#PTP_PARAMS,12)
PTP XPlace_R1_L6_S1_VP3 C_DIS
;ENDFOLD
TRIGGER WHEN DISTANCE=1 DELAY=-1 DO Schrittmerker_R1Place(10613,10612,FPlace_R1_L6_S1_VP4,XPlace_R1_L6_S1_VP4) PRIO=-1
;FOLD PTP Place_R1_L6_S1_VP4 CONT Vel=12 % PPlace_R1_L6_S1_VP4 Tool[1]:Upper Gripper Base[0];%{PE}%R8.3.21,%MKUKATPBASIS,%CMOVE,%VPTP,%P 1:PTP, 2:Place_R1_L6_S1_VP4, 3:C_DIS, 5:12, 7:PPlace_R1_L6_S1_VP4
$BWDSTART=FALSE
PDAT_ACT= PPPlace_R1_L6_S1_VP4
FDAT_ACT= FPlace_R1_L6_S1_VP4
BAS(#PTP_PARAMS,12)
PTP XPlace_R1_L6_S1_VP4 C_DIS
;ENDFOLD
TRIGGER WHEN DISTANCE=1 DELAY=-1 DO Schrittmerker_R1Place(10614,10613,FPlace_R1_L6_S1_VP5,XPlace_R1_L6_S1_VP5) PRIO=-1
;FOLD PTP Place_R1_L6_S1_VP5 CONT Vel=12 % PPlace_R1_L6_S1_VP5 Tool[1]:Upper Gripper Base[0];%{PE}%R8.3.21,%MKUKATPBASIS,%CMOVE,%VPTP,%P 1:PTP, 2:Place_R1_L6_S1_VP5, 3:C_DIS, 5:12, 7:PPlace_R1_L6_S1_VP5
$BWDSTART=FALSE
PDAT_ACT= PPPlace_R1_L6_S1_VP5
FDAT_ACT= FPlace_R1_L6_S1_VP5
BAS(#PTP_PARAMS,12)
PTP XPlace_R1_L6_S1_VP5 C_DIS
;ENDFOLD
TRIGGER WHEN DISTANCE=1 DELAY=-1 DO Schrittmerker_R1Place(10615,10614,FPlace_R1_L6_S1_VP6,XPlace_R1_L6_S1_VP6) PRIO=-1
;FOLD PTP Place_R1_L6_S1_VP6 CONT Vel=12 % PPlace_R1_L6_S1_VP6 Tool[1]:Upper Gripper Base[0];%{PE}%R8.3.21,%MKUKATPBASIS,%CMOVE,%VPTP,%P 1:PTP, 2:Place_R1_L6_S1_VP6, 3:C_DIS, 5:12, 7:PPlace_R1_L6_S1_VP6
$BWDSTART=FALSE
PDAT_ACT= PPPlace_R1_L6_S1_VP6
FDAT_ACT= FPlace_R1_L6_S1_VP6
BAS(#PTP_PARAMS,12)
PTP XPlace_R1_L6_S1_VP6 C_DIS
;ENDFOLD
TRIGGER WHEN DISTANCE=1 DELAY=-1 DO Schrittmerker_R1Place(10616,10615,FPlace_R1_L6_S1_VP7,XPlace_R1_L6_S1_VP7) PRIO=-1
;FOLD PTP Place_R1_L6_S1_VP7 CONT Vel=12 % PPlace_R1_L6_S1_VP7 Tool[1]:Upper Gripper Base[0];%{PE}%R8.3.21,%MKUKATPBASIS,%CMOVE,%VPTP,%P 1:PTP, 2:Place_R1_L6_S1_VP7, 3:C_DIS, 5:12, 7:PPlace_R1_L6_S1_VP7
$BWDSTART=FALSE
PDAT_ACT= PPPlace_R1_L6_S1_VP7
FDAT_ACT= FPlace_R1_L6_S1_VP7
BAS(#PTP_PARAMS,12)
PTP XPlace_R1_L6_S1_VP7 C_DIS
;ENDFOLD
TRIGGER WHEN DISTANCE=1 DELAY=-1 DO Schrittmerker_R1Place(10617,10616,FPlace_R1_L6_S1_VP8,XPlace_R1_L6_S1_VP8) PRIO=-1
;FOLD PTP Place_R1_L6_S1_VP8 CONT Vel=12 % PPlace_R1_L6_S1_VP8 Tool[1]:Upper Gripper Base[0];%{PE}%R8.3.21,%MKUKATPBASIS,%CMOVE,%VPTP,%P 1:PTP, 2:Place_R1_L6_S1_VP8, 3:C_DIS, 5:12, 7:PPlace_R1_L6_S1_VP8
$BWDSTART=FALSE
PDAT_ACT= PPPlace_R1_L6_S1_VP8
FDAT_ACT= FPlace_R1_L6_S1_VP8
BAS(#PTP_PARAMS,12)
PTP XPlace_R1_L6_S1_VP8 C_DIS
;ENDFOLD

TRIGGER WHEN DISTANCE=1 DELAY=-1 DO Schrittmerker_R1Place(10618,10617,FPlace_R1_L6_S1_Check,XPlace_R1_L6_S1_Check) PRIO=-1
;FOLD PTP Place_R1_L6_S1_Check Vel=12 % PPlace_R1_L6_S1_Check Tool[1]:Upper Gripper Base[1]:Rack1;%{PE}%R8.3.21,%MKUKATPBASIS,%CMOVE,%VPTP,%P 1:PTP, 2:Place_R1_L6_S1_Check, 3:, 5:12, 7:PPlace_R1_L6_S1_Check
$BWDSTART=FALSE
PDAT_ACT= PPPlace_R1_L6_S1_Check
FDAT_ACT= FPlace_R1_L6_S1_Check
BAS(#PTP_PARAMS,12)
PTP XPlace_R1_L6_S1_Check
;ENDFOLD

;***************************************************
;FOLD Pruefe Platz frei
IF (DetectPart(CHECK_SHELF,PLACE)==OCCUPIED) THEN
  UP_Rueckzug_R1Place( )
  RETURN
ENDIF
;ENDFOLD
;***************************************************

TRIGGER WHEN DISTANCE=1 DELAY=-1 DO Schrittmerker_R1Place(10619,10618,FPlace_R1_L6_S1_VP9,XPlace_R1_L6_S1_VP9) PRIO=-1
;FOLD LIN Place_R1_L6_S1_VP9 CONT Vel=0.5 m/s LPlace_R1_L6_S1_VP9 Tool[1]:Upper Gripper Base[1]:Rack1;%{PE}%R8.3.21,%MKUKATPBASIS,%CMOVE,%VLIN,%P 1:LIN, 2:Place_R1_L6_S1_VP9, 3:C_DIS C_DIS, 5:0.5, 7:LPlace_R1_L6_S1_VP9
$BWDSTART=FALSE
LDAT_ACT= LLPlace_R1_L6_S1_VP9
FDAT_ACT= FPlace_R1_L6_S1_VP9
BAS(#CP_PARAMS,0.5)
LIN XPlace_R1_L6_S1_VP9 C_DIS C_DIS
;ENDFOLD
TRIGGER WHEN DISTANCE=1 DELAY=-1 DO Schrittmerker_R1Place(10620,10619,FPlace_R1_L6_S1_VP10,XPlace_R1_L6_S1_VP10) PRIO=-1
;FOLD LIN Place_R1_L6_S1_VP10 CONT Vel=0.5 m/s LPlace_R1_L6_S1_VP10 Tool[1]:Upper Gripper Base[1]:Rack1;%{PE}%R8.3.21,%MKUKATPBASIS,%CMOVE,%VLIN,%P 1:LIN, 2:Place_R1_L6_S1_VP10, 3:C_DIS C_DIS, 5:0.5, 7:LPlace_R1_L6_S1_VP10
$BWDSTART=FALSE
LDAT_ACT= LLPlace_R1_L6_S1_VP10
FDAT_ACT= FPlace_R1_L6_S1_VP10
BAS(#CP_PARAMS,0.5)
LIN XPlace_R1_L6_S1_VP10 C_DIS C_DIS
;ENDFOLD
TRIGGER WHEN DISTANCE=1 DELAY=-1 DO Schrittmerker_R1Place(10621,10620,FPlace_R1_L6_S1_VP11,XPlace_R1_L6_S1_VP11) PRIO=-1
;FOLD LIN Place_R1_L6_S1_VP11 CONT Vel=0.5 m/s LPlace_R1_L6_S1_VP11 Tool[1]:Upper Gripper Base[1]:Rack1;%{PE}%R8.3.21,%MKUKATPBASIS,%CMOVE,%VLIN,%P 1:LIN, 2:Place_R1_L6_S1_VP11, 3:C_DIS C_DIS, 5:0.5, 7:LPlace_R1_L6_S1_VP11
$BWDSTART=FALSE
LDAT_ACT= LLPlace_R1_L6_S1_VP11
FDAT_ACT= FPlace_R1_L6_S1_VP11
BAS(#CP_PARAMS,0.5)
LIN XPlace_R1_L6_S1_VP11 C_DIS C_DIS
;ENDFOLD

;FOLD Test the way back home - part 1
CONTINUE
IF ($FLAG[M_Test_GrdstFahren1] AND NOT $FLAG[M_Test_GrdstFahren2]) THEN
  $FLAG[M_Test_GrdstFahren2]=TRUE
  UP_Rueckzug( )
  RETURN
ENDIF
;ENDFOLD

;-------------------------------
; Place part position
;-------------------------------
TRIGGER WHEN DISTANCE=1 DELAY=-1 DO Schrittmerker_R1Place(10622,10623,FPlace_R1_L6_S1_AP,XPlace_R1_L6_S1_AP) PRIO=-1
;FOLD LIN Place_R1_L6_S1_AP Vel=0.2 m/s LPlace_R1_L6_S1_AP Tool[1]:Upper Gripper Base[1]:Rack1;%{PE}%R8.3.21,%MKUKATPBASIS,%CMOVE,%VLIN,%P 1:LIN, 2:Place_R1_L6_S1_AP, 3:, 5:0.2, 7:LPlace_R1_L6_S1_AP
$BWDSTART=FALSE
LDAT_ACT= LLPlace_R1_L6_S1_AP
FDAT_ACT= FPlace_R1_L6_S1_AP
BAS(#CP_PARAMS,0.2)
LIN XPlace_R1_L6_S1_AP
;ENDFOLD

;FOLD Test the way back home - part 2
CONTINUE
IF $FLAG[M_Test_GrdstFahren2] THEN
  $FLAG[M_Test_GrdstFahren2]=FALSE
  UP_Rueckzug( )
  RETURN
ENDIF
;ENDFOLD

;***************************************************
; Disable part lost detection
SetPartLostDetection(NO_PART)
;***************************************************

TRIGGER WHEN DISTANCE=1 DELAY=-1 DO Schrittmerker_R1Place(10623,10624,FPlace_R1_L6_S1_NP1,XPlace_R1_L6_S1_NP1) PRIO=-1
;FOLD LIN Place_R1_L6_S1_NP1 Vel=0.2 m/s LPlace_R1_L6_S1_NP1 Tool[1]:Upper Gripper Base[1]:Rack1;%{PE}%R8.3.21,%MKUKATPBASIS,%CMOVE,%VLIN,%P 1:LIN, 2:Place_R1_L6_S1_NP1, 3:C_DIS C_DIS, 5:0.2, 7:LPlace_R1_L6_S1_NP1
$BWDSTART=FALSE
LDAT_ACT= LLPlace_R1_L6_S1_NP1
FDAT_ACT= FPlace_R1_L6_S1_NP1
BAS(#CP_PARAMS,0.2)
LIN XPlace_R1_L6_S1_NP1
;ENDFOLD

;***************************************************
; Check for part present (empty gripper)
CheckPartPresent(EMPTY_GRIPPER)
;***************************************************
; set load data
SetLoadData( )
;***************************************************

TRIGGER WHEN DISTANCE=1 DELAY=-1 DO Schrittmerker_R1Place(10624,10625,FPlace_R1_L6_S1_NP2,XPlace_R1_L6_S1_NP2) PRIO=-1
;FOLD LIN Place_R1_L6_S1_NP2 CONT Vel=0.5 m/s LPlace_R1_L6_S1_NP2 Tool[1]:Upper Gripper Base[1]:Rack1;%{PE}%R8.3.21,%MKUKATPBASIS,%CMOVE,%VLIN,%P 1:LIN, 2:Place_R1_L6_S1_NP2, 3:C_DIS C_DIS, 5:0.5, 7:LPlace_R1_L6_S1_NP2
$BWDSTART=FALSE
LDAT_ACT= LLPlace_R1_L6_S1_NP2
FDAT_ACT= FPlace_R1_L6_S1_NP2
BAS(#CP_PARAMS,0.5)
LIN XPlace_R1_L6_S1_NP2 C_DIS C_DIS
;ENDFOLD
TRIGGER WHEN DISTANCE=1 DELAY=-1 DO Schrittmerker_R1Place(10625,10626,FPlace_R1_L6_S1_NP3,XPlace_R1_L6_S1_NP3) PRIO=-1
;FOLD LIN Place_R1_L6_S1_NP3 Vel=0.5 m/s LPlace_R1_L6_S1_NP3 Tool[1]:Upper Gripper Base[1]:Rack1;%{PE}%R8.3.21,%MKUKATPBASIS,%CMOVE,%VLIN,%P 1:LIN, 2:Place_R1_L6_S1_NP3, 3:, 5:0.5, 7:LPlace_R1_L6_S1_NP3
$BWDSTART=FALSE
LDAT_ACT= LLPlace_R1_L6_S1_NP3
FDAT_ACT= FPlace_R1_L6_S1_NP3
BAS(#CP_PARAMS,0.5)
LIN XPlace_R1_L6_S1_NP3
;ENDFOLD
TRIGGER WHEN DISTANCE=1 DELAY=-1 DO Schrittmerker_R1Place(10626,10627,FPlace_R1_L6_S1_NP4,XPlace_R1_L6_S1_NP4) PRIO=-1
;FOLD PTP Place_R1_L6_S1_NP4 CONT Vel=100 % PPlace_R1_L6_S1_NP4 Tool[1]:Upper Gripper Base[1]:Rack1;%{PE}%R8.3.21,%MKUKATPBASIS,%CMOVE,%VPTP,%P 1:PTP, 2:Place_R1_L6_S1_NP4, 3:C_DIS, 5:100, 7:PPlace_R1_L6_S1_NP4
$BWDSTART=FALSE
PDAT_ACT= PPPlace_R1_L6_S1_NP4
FDAT_ACT= FPlace_R1_L6_S1_NP4
BAS(#PTP_PARAMS,100)
PTP XPlace_R1_L6_S1_NP4 C_DIS
;ENDFOLD
TRIGGER WHEN DISTANCE=1 DELAY=-1 DO Schrittmerker_R1Place(10627,10628,FPlace_R1_L6_S1_NP5,XPlace_R1_L6_S1_NP5) PRIO=-1
;FOLD PTP Place_R1_L6_S1_NP5 CONT Vel=100 % PPlace_R1_L6_S1_NP5 Tool[1]:Upper Gripper Base[0];%{PE}%R8.3.21,%MKUKATPBASIS,%CMOVE,%VPTP,%P 1:PTP, 2:Place_R1_L6_S1_NP5, 3:C_DIS, 5:100, 7:PPlace_R1_L6_S1_NP5
$BWDSTART=FALSE
PDAT_ACT= PPPlace_R1_L6_S1_NP5
FDAT_ACT= FPlace_R1_L6_S1_NP5
BAS(#PTP_PARAMS,100)
PTP XPlace_R1_L6_S1_NP5 C_DIS
;ENDFOLD
TRIGGER WHEN DISTANCE=1 DELAY=-1 DO Schrittmerker_R1Place(10628,10629,FPlace_R1_L6_S1_NP6,XPlace_R1_L6_S1_NP6) PRIO=-1
;FOLD PTP Place_R1_L6_S1_NP6 CONT Vel=100 % PPlace_R1_L6_S1_NP6 Tool[1]:Upper Gripper Base[0];%{PE}%R8.3.21,%MKUKATPBASIS,%CMOVE,%VPTP,%P 1:PTP, 2:Place_R1_L6_S1_NP6, 3:C_DIS, 5:100, 7:PPlace_R1_L6_S1_NP6
$BWDSTART=FALSE
PDAT_ACT= PPPlace_R1_L6_S1_NP6
FDAT_ACT= FPlace_R1_L6_S1_NP6
BAS(#PTP_PARAMS,100)
PTP XPlace_R1_L6_S1_NP6 C_DIS
;ENDFOLD
TRIGGER WHEN DISTANCE=1 DELAY=-1 DO Schrittmerker_R1Place(10629,10630,FPlace_R1_L6_S1_NP7,XPlace_R1_L6_S1_NP7) PRIO=-1
;FOLD PTP Place_R1_L6_S1_NP7 CONT Vel=100 % PPlace_R1_L6_S1_NP7 Tool[1]:Upper Gripper Base[0];%{PE}%R8.3.21,%MKUKATPBASIS,%CMOVE,%VPTP,%P 1:PTP, 2:Place_R1_L6_S1_NP7, 3:C_DIS, 5:100, 7:PPlace_R1_L6_S1_NP7
$BWDSTART=FALSE
PDAT_ACT= PPPlace_R1_L6_S1_NP7
FDAT_ACT= FPlace_R1_L6_S1_NP7
BAS(#PTP_PARAMS,100)
PTP XPlace_R1_L6_S1_NP7 C_DIS
;ENDFOLD

TRIGGER WHEN DISTANCE=1 DELAY=-1 DO Schrittmerker_R1Place(10630,10501,FHOME,$nullframe,XHOME) PRIO=-1
;FOLD PTP HOME Vel=100 % PHome;%{PE}%R8.3.21,%MKUKATPBASIS,%CMOVE,%VPTP,%P 1:PTP, 2:HOME, 3:, 5:100, 7:PHome
$BWDSTART=FALSE
PDAT_ACT= PPHome
FDAT_ACT= FHOME
BAS(#PTP_PARAMS,100)
PTP XHOME
;ENDFOLD

;***************************************************
;FOLD Final tasks.
; Robot out of area Rack 1 Level 6
RobAusStorage1_6_A72=RESET_IN_AREA
;***************************************************
; stop cyclic clearence check
$CYCFLAG[ciFreigabeSPS]=DISABLE_MONITORING
;***************************************************
; Disable collision detection
;FOLD COLLDETECT Off ;%{PE}
;FOLD Parameters ;%{h}
;Params IlfProvider=kukaroboter.basistech.inlineforms.colldetect.off; CollDetect.Command=Off
;ENDFOLD
USE_CD_PARAMS(0)
;ENDFOLD
;***************************************************
;ENDFOLD
;***************************************************

END

; ##################################################

GLOBAL DEF UP_Place_R1_L6_S2( )
;***************************************************
; Place part on:
;    Rack  1
;    Level 6
;    Shelf 2
;***************************************************
;FOLD Preconditions - Vorraussetzungen
;***************************************************
; Enable collision detection
;FOLD COLLDETECT SetLimits Axis1: 150 % Axis2: 200 % Axis3: 150 % Axis4: 200 % Axis5: 150 % Axis6: 150 % ;%{PE}
;FOLD Parameters ;%{h}
;Params IlfProvider=kukaroboter.basistech.inlineforms.colldetect.setlimits; CollDetect.Command=SetLimits; CollDetect.Axis1=150; CollDetect.Axis2=200; CollDetect.Axis3=150; CollDetect.Axis4=200; CollDetect.Axis5=150; CollDetect.Axis6=150
;ENDFOLD
SET_TQ_VALUES(150, 200, 150, 200, 150, 150)
;ENDFOLD
;***************************************************
; Check for part in gripper (tool 1).
CheckPartPresent(OCCUPIED_GRIPPER,PART_ON_TOOL_1)
;***************************************************
; Enable part lost detection for tool 1
SetPartLostDetection(PART_ON_TOOL_1)
;***************************************************
; Set load data.
SetLoadData( )
;***************************************************
; Robot has to start from home position.
IF NOT $IN_HOME THEN
  UP_HomeToHome(0)
ENDIF
;***************************************************
;ENDFOLD

TRIGGER WHEN DISTANCE=1 DELAY=-1 DO Schrittmerker_R1Place(10501,10501,FHOME,$nullframe,XHOME) PRIO=-1
;FOLD PTP HOME Vel=12 % PHome;%{PE}%R8.3.21,%MKUKATPBASIS,%CMOVE,%VPTP,%P 1:PTP, 2:HOME, 3:, 5:12, 7:PHome
$BWDSTART=FALSE
PDAT_ACT= PPHome
FDAT_ACT= FHOME
BAS(#PTP_PARAMS,12)
PTP XHOME
;ENDFOLD

;***************************************************
;FOLD Area clearence handshake.
IF NOT $FLAG[M_Inbetriebnahme] THEN
  ;-------------------------------------------------
  ; Request area clearence.
  AnfStoer_Store1_6_A104=SET_REQUEST
  ;-------------------------------------------------
  ; Wait for area clearence from PLC.
  WAIT_FOR_INPUT("Frg_Storage1_6_E72",TRUE)
  ;-------------------------------------------------
  ; Reset area clearence request.
  AnfStoer_Store1_6_A104=RESET_REQUEST
  ;-------------------------------------------------
  ; start cyclic clearence check
  $CYCFLAG[ciFreigabeSPS]=Frg_Storage1_6_E72
  ;-------------------------------------------------
ENDIF
;***************************************************
; set "robot in area"
RobAusStorage1_6_A72=SET_IN_AREA
;ENDFOLD
;***************************************************

;***************************************************
;FOLD Check for Teachmode
IF $FLAG[M_Teachen] THEN
  WAIT FOR $T1
ENDIF
;ENDFOLD
;***************************************************

; move to the rack
TRIGGER WHEN DISTANCE=1 DELAY=-1 DO Schrittmerker_R1Place(10640,10501,FPlace_R1_L6_S2_VP1,XPlace_R1_L6_S2_VP1) PRIO=-1
;FOLD PTP Place_R1_L6_S2_VP1 CONT Vel=12 % PPlace_R1_L6_S2_VP1 Tool[1]:Upper Gripper Base[0];%{PE}%R8.3.21,%MKUKATPBASIS,%CMOVE,%VPTP,%P 1:PTP, 2:Place_R1_L6_S2_VP1, 3:C_DIS, 5:12, 7:PPlace_R1_L6_S2_VP1
$BWDSTART=FALSE
PDAT_ACT= PPPlace_R1_L6_S2_VP1
FDAT_ACT= FPlace_R1_L6_S2_VP1
BAS(#PTP_PARAMS,12)
PTP XPlace_R1_L6_S2_VP1 C_DIS
;ENDFOLD
TRIGGER WHEN DISTANCE=1 DELAY=-1 DO Schrittmerker_R1Place(10641,10640,FPlace_R1_L6_S2_VP2,XPlace_R1_L6_S2_VP2) PRIO=-1
;FOLD PTP Place_R1_L6_S2_VP2 CONT Vel=12 % PPlace_R1_L6_S2_VP2 Tool[1]:Upper Gripper Base[0];%{PE}%R8.3.21,%MKUKATPBASIS,%CMOVE,%VPTP,%P 1:PTP, 2:Place_R1_L6_S2_VP2, 3:C_DIS, 5:12, 7:PPlace_R1_L6_S2_VP2
$BWDSTART=FALSE
PDAT_ACT= PPPlace_R1_L6_S2_VP2
FDAT_ACT= FPlace_R1_L6_S2_VP2
BAS(#PTP_PARAMS,12)
PTP XPlace_R1_L6_S2_VP2 C_DIS
;ENDFOLD
TRIGGER WHEN DISTANCE=1 DELAY=-1 DO Schrittmerker_R1Place(10642,10641,FPlace_R1_L6_S2_VP3,XPlace_R1_L6_S2_VP3) PRIO=-1
;FOLD PTP Place_R1_L6_S2_VP3 CONT Vel=12 % PPlace_R1_L6_S2_VP3 Tool[1]:Upper Gripper Base[0];%{PE}%R8.3.21,%MKUKATPBASIS,%CMOVE,%VPTP,%P 1:PTP, 2:Place_R1_L6_S2_VP3, 3:C_DIS, 5:12, 7:PPlace_R1_L6_S2_VP3
$BWDSTART=FALSE
PDAT_ACT= PPPlace_R1_L6_S2_VP3
FDAT_ACT= FPlace_R1_L6_S2_VP3
BAS(#PTP_PARAMS,12)
PTP XPlace_R1_L6_S2_VP3 C_DIS
;ENDFOLD
TRIGGER WHEN DISTANCE=1 DELAY=-1 DO Schrittmerker_R1Place(10643,10642,FPlace_R1_L6_S2_VP4,XPlace_R1_L6_S2_VP4) PRIO=-1
;FOLD PTP Place_R1_L6_S2_VP4 CONT Vel=12 % PPlace_R1_L6_S2_VP4 Tool[1]:Upper Gripper Base[0];%{PE}%R8.3.21,%MKUKATPBASIS,%CMOVE,%VPTP,%P 1:PTP, 2:Place_R1_L6_S2_VP4, 3:C_DIS, 5:12, 7:PPlace_R1_L6_S2_VP4
$BWDSTART=FALSE
PDAT_ACT= PPPlace_R1_L6_S2_VP4
FDAT_ACT= FPlace_R1_L6_S2_VP4
BAS(#PTP_PARAMS,12)
PTP XPlace_R1_L6_S2_VP4 C_DIS
;ENDFOLD
TRIGGER WHEN DISTANCE=1 DELAY=-1 DO Schrittmerker_R1Place(10644,10643,FPlace_R1_L6_S2_VP5,XPlace_R1_L6_S2_VP5) PRIO=-1
;FOLD PTP Place_R1_L6_S2_VP5 CONT Vel=12 % PPlace_R1_L6_S2_VP5 Tool[1]:Upper Gripper Base[0];%{PE}%R8.3.21,%MKUKATPBASIS,%CMOVE,%VPTP,%P 1:PTP, 2:Place_R1_L6_S2_VP5, 3:C_DIS, 5:12, 7:PPlace_R1_L6_S2_VP5
$BWDSTART=FALSE
PDAT_ACT= PPPlace_R1_L6_S2_VP5
FDAT_ACT= FPlace_R1_L6_S2_VP5
BAS(#PTP_PARAMS,12)
PTP XPlace_R1_L6_S2_VP5 C_DIS
;ENDFOLD
TRIGGER WHEN DISTANCE=1 DELAY=-1 DO Schrittmerker_R1Place(10645,10644,FPlace_R1_L6_S2_VP6,XPlace_R1_L6_S2_VP6) PRIO=-1
;FOLD PTP Place_R1_L6_S2_VP6 CONT Vel=12 % PPlace_R1_L6_S2_VP6 Tool[1]:Upper Gripper Base[0];%{PE}%R8.3.21,%MKUKATPBASIS,%CMOVE,%VPTP,%P 1:PTP, 2:Place_R1_L6_S2_VP6, 3:C_DIS, 5:12, 7:PPlace_R1_L6_S2_VP6
$BWDSTART=FALSE
PDAT_ACT= PPPlace_R1_L6_S2_VP6
FDAT_ACT= FPlace_R1_L6_S2_VP6
BAS(#PTP_PARAMS,12)
PTP XPlace_R1_L6_S2_VP6 C_DIS
;ENDFOLD
TRIGGER WHEN DISTANCE=1 DELAY=-1 DO Schrittmerker_R1Place(10646,10645,FPlace_R1_L6_S2_VP7,XPlace_R1_L6_S2_VP7) PRIO=-1
;FOLD PTP Place_R1_L6_S2_VP7 CONT Vel=12 % PPlace_R1_L6_S2_VP7 Tool[1]:Upper Gripper Base[0];%{PE}%R8.3.21,%MKUKATPBASIS,%CMOVE,%VPTP,%P 1:PTP, 2:Place_R1_L6_S2_VP7, 3:C_DIS, 5:12, 7:PPlace_R1_L6_S2_VP7
$BWDSTART=FALSE
PDAT_ACT= PPPlace_R1_L6_S2_VP7
FDAT_ACT= FPlace_R1_L6_S2_VP7
BAS(#PTP_PARAMS,12)
PTP XPlace_R1_L6_S2_VP7 C_DIS
;ENDFOLD
TRIGGER WHEN DISTANCE=1 DELAY=-1 DO Schrittmerker_R1Place(10647,10646,FPlace_R1_L6_S2_VP8,XPlace_R1_L6_S2_VP8) PRIO=-1
;FOLD PTP Place_R1_L6_S2_VP8 CONT Vel=12 % PPlace_R1_L6_S2_VP8 Tool[1]:Upper Gripper Base[1]:Rack1;%{PE}%R8.3.21,%MKUKATPBASIS,%CMOVE,%VPTP,%P 1:PTP, 2:Place_R1_L6_S2_VP8, 3:C_DIS, 5:12, 7:PPlace_R1_L6_S2_VP8
$BWDSTART=FALSE
PDAT_ACT= PPPlace_R1_L6_S2_VP8
FDAT_ACT= FPlace_R1_L6_S2_VP8
BAS(#PTP_PARAMS,12)
PTP XPlace_R1_L6_S2_VP8 C_DIS
;ENDFOLD

TRIGGER WHEN DISTANCE=1 DELAY=-1 DO Schrittmerker_R1Place(10648,10647,FPlace_R1_L6_S2_Check,XPlace_R1_L6_S2_Check) PRIO=-1
;FOLD PTP Place_R1_L6_S2_Check Vel=12 % PPlace_R1_L6_S2_Check Tool[1]:Upper Gripper Base[1]:Rack1;%{PE}%R8.3.21,%MKUKATPBASIS,%CMOVE,%VPTP,%P 1:PTP, 2:Place_R1_L6_S2_Check, 3:, 5:12, 7:PPlace_R1_L6_S2_Check
$BWDSTART=FALSE
PDAT_ACT= PPPlace_R1_L6_S2_Check
FDAT_ACT= FPlace_R1_L6_S2_Check
BAS(#PTP_PARAMS,12)
PTP XPlace_R1_L6_S2_Check
;ENDFOLD

;***************************************************
;FOLD Pruefe Platz frei
IF (DetectPart(CHECK_SHELF,PLACE)==OCCUPIED) THEN
  UP_Rueckzug_R1Place( )
  RETURN
ENDIF
;ENDFOLD
;***************************************************

TRIGGER WHEN DISTANCE=1 DELAY=-1 DO Schrittmerker_R1Place(10649,10648,FPlace_R1_L6_S2_VP9,XPlace_R1_L6_S2_VP9) PRIO=-1
;FOLD LIN Place_R1_L6_S2_VP9 CONT Vel=0.5 m/s LPlace_R1_L6_S2_VP9 Tool[1]:Upper Gripper Base[1]:Rack1;%{PE}%R8.3.21,%MKUKATPBASIS,%CMOVE,%VLIN,%P 1:LIN, 2:Place_R1_L6_S2_VP9, 3:C_DIS C_DIS, 5:0.5, 7:LPlace_R1_L6_S2_VP9
$BWDSTART=FALSE
LDAT_ACT= LLPlace_R1_L6_S2_VP9
FDAT_ACT= FPlace_R1_L6_S2_VP9
BAS(#CP_PARAMS,0.5)
LIN XPlace_R1_L6_S2_VP9 C_DIS C_DIS
;ENDFOLD
TRIGGER WHEN DISTANCE=1 DELAY=-1 DO Schrittmerker_R1Place(10650,10649,FPlace_R1_L6_S2_VP10,XPlace_R1_L6_S2_VP10) PRIO=-1
;FOLD LIN Place_R1_L6_S2_VP10 CONT Vel=0.5 m/s LPlace_R1_L6_S2_VP10 Tool[1]:Upper Gripper Base[1]:Rack1;%{PE}%R8.3.21,%MKUKATPBASIS,%CMOVE,%VLIN,%P 1:LIN, 2:Place_R1_L6_S2_VP10, 3:C_DIS C_DIS, 5:0.5, 7:LPlace_R1_L6_S2_VP10
$BWDSTART=FALSE
LDAT_ACT= LLPlace_R1_L6_S2_VP10
FDAT_ACT= FPlace_R1_L6_S2_VP10
BAS(#CP_PARAMS,0.5)
LIN XPlace_R1_L6_S2_VP10 C_DIS C_DIS
;ENDFOLD
TRIGGER WHEN DISTANCE=1 DELAY=-1 DO Schrittmerker_R1Place(10651,10650,FPlace_R1_L6_S2_VP11,XPlace_R1_L6_S2_VP11) PRIO=-1
;FOLD LIN Place_R1_L6_S2_VP11 CONT Vel=0.5 m/s LPlace_R1_L6_S2_VP11 Tool[1]:Upper Gripper Base[1]:Rack1;%{PE}%R8.3.21,%MKUKATPBASIS,%CMOVE,%VLIN,%P 1:LIN, 2:Place_R1_L6_S2_VP11, 3:C_DIS C_DIS, 5:0.5, 7:LPlace_R1_L6_S2_VP11
$BWDSTART=FALSE
LDAT_ACT= LLPlace_R1_L6_S2_VP11
FDAT_ACT= FPlace_R1_L6_S2_VP11
BAS(#CP_PARAMS,0.5)
LIN XPlace_R1_L6_S2_VP11 C_DIS C_DIS
;ENDFOLD

;FOLD Test the way back home - part 1
CONTINUE
IF ($FLAG[M_Test_GrdstFahren1] AND NOT $FLAG[M_Test_GrdstFahren2]) THEN
  $FLAG[M_Test_GrdstFahren2]=TRUE
  UP_Rueckzug( )
  RETURN
ENDIF
;ENDFOLD

;-------------------------------
; Place part position
;-------------------------------
TRIGGER WHEN DISTANCE=1 DELAY=-1 DO Schrittmerker_R1Place(10652,10653,FPlace_R1_L6_S2_AP,XPlace_R1_L6_S2_AP) PRIO=-1
;FOLD LIN Place_R1_L6_S2_AP Vel=0.2 m/s LPlace_R1_L6_S2_AP Tool[1]:Upper Gripper Base[1]:Rack1;%{PE}%R8.3.21,%MKUKATPBASIS,%CMOVE,%VLIN,%P 1:LIN, 2:Place_R1_L6_S2_AP, 3:, 5:0.2, 7:LPlace_R1_L6_S2_AP
$BWDSTART=FALSE
LDAT_ACT= LLPlace_R1_L6_S2_AP
FDAT_ACT= FPlace_R1_L6_S2_AP
BAS(#CP_PARAMS,0.2)
LIN XPlace_R1_L6_S2_AP
;ENDFOLD

;FOLD Test the way back home - part 2
CONTINUE
IF $FLAG[M_Test_GrdstFahren2] THEN
  $FLAG[M_Test_GrdstFahren2]=FALSE
  UP_Rueckzug( )
  RETURN
ENDIF
;ENDFOLD

;***************************************************
; Disable part lost detection
SetPartLostDetection(NO_PART)
;***************************************************

TRIGGER WHEN DISTANCE=1 DELAY=-1 DO Schrittmerker_R1Place(10653,10654,FPlace_R1_L6_S2_NP1,XPlace_R1_L6_S2_NP1) PRIO=-1
;FOLD LIN Place_R1_L6_S2_NP1 Vel=0.2 m/s LPlace_R1_L6_S2_NP1 Tool[1]:Upper Gripper Base[1]:Rack1;%{PE}%R8.3.21,%MKUKATPBASIS,%CMOVE,%VLIN,%P 1:LIN, 2:Place_R1_L6_S2_NP1, 3:C_DIS C_DIS, 5:0.2, 7:LPlace_R1_L6_S2_NP1
$BWDSTART=FALSE
LDAT_ACT= LLPlace_R1_L6_S2_NP1
FDAT_ACT= FPlace_R1_L6_S2_NP1
BAS(#CP_PARAMS,0.2)
LIN XPlace_R1_L6_S2_NP1
;ENDFOLD

;***************************************************
; Check for part present (empty gripper)
CheckPartPresent(EMPTY_GRIPPER)
;***************************************************
; set load data
SetLoadData( )
;***************************************************

TRIGGER WHEN DISTANCE=1 DELAY=-1 DO Schrittmerker_R1Place(10654,10655,FPlace_R1_L6_S2_NP2,XPlace_R1_L6_S2_NP2) PRIO=-1
;FOLD LIN Place_R1_L6_S2_NP2 CONT Vel=0.5 m/s LPlace_R1_L6_S2_NP2 Tool[1]:Upper Gripper Base[1]:Rack1;%{PE}%R8.3.21,%MKUKATPBASIS,%CMOVE,%VLIN,%P 1:LIN, 2:Place_R1_L6_S2_NP2, 3:C_DIS C_DIS, 5:0.5, 7:LPlace_R1_L6_S2_NP2
$BWDSTART=FALSE
LDAT_ACT= LLPlace_R1_L6_S2_NP2
FDAT_ACT= FPlace_R1_L6_S2_NP2
BAS(#CP_PARAMS,0.5)
LIN XPlace_R1_L6_S2_NP2 C_DIS C_DIS
;ENDFOLD
TRIGGER WHEN DISTANCE=1 DELAY=-1 DO Schrittmerker_R1Place(10655,10656,FPlace_R1_L6_S2_NP3,XPlace_R1_L6_S2_NP3) PRIO=-1
;FOLD LIN Place_R1_L6_S2_NP3 Vel=0.5 m/s LPlace_R1_L6_S2_NP3 Tool[1]:Upper Gripper Base[1]:Rack1;%{PE}%R8.3.21,%MKUKATPBASIS,%CMOVE,%VLIN,%P 1:LIN, 2:Place_R1_L6_S2_NP3, 3:, 5:0.5, 7:LPlace_R1_L6_S2_NP3
$BWDSTART=FALSE
LDAT_ACT= LLPlace_R1_L6_S2_NP3
FDAT_ACT= FPlace_R1_L6_S2_NP3
BAS(#CP_PARAMS,0.5)
LIN XPlace_R1_L6_S2_NP3
;ENDFOLD
TRIGGER WHEN DISTANCE=1 DELAY=-1 DO Schrittmerker_R1Place(10656,10657,FPlace_R1_L6_S2_NP4,XPlace_R1_L6_S2_NP4) PRIO=-1
;FOLD PTP Place_R1_L6_S2_NP4 CONT Vel=100 % PPlace_R1_L6_S2_NP4 Tool[1]:Upper Gripper Base[1]:Rack1;%{PE}%R8.3.21,%MKUKATPBASIS,%CMOVE,%VPTP,%P 1:PTP, 2:Place_R1_L6_S2_NP4, 3:C_DIS, 5:100, 7:PPlace_R1_L6_S2_NP4
$BWDSTART=FALSE
PDAT_ACT= PPPlace_R1_L6_S2_NP4
FDAT_ACT= FPlace_R1_L6_S2_NP4
BAS(#PTP_PARAMS,100)
PTP XPlace_R1_L6_S2_NP4 C_DIS
;ENDFOLD
TRIGGER WHEN DISTANCE=1 DELAY=-1 DO Schrittmerker_R1Place(10657,10658,FPlace_R1_L6_S2_NP5,XPlace_R1_L6_S2_NP5) PRIO=-1
;FOLD PTP Place_R1_L6_S2_NP5 CONT Vel=100 % PPlace_R1_L6_S2_NP5 Tool[1]:Upper Gripper Base[0];%{PE}%R8.3.21,%MKUKATPBASIS,%CMOVE,%VPTP,%P 1:PTP, 2:Place_R1_L6_S2_NP5, 3:C_DIS, 5:100, 7:PPlace_R1_L6_S2_NP5
$BWDSTART=FALSE
PDAT_ACT= PPPlace_R1_L6_S2_NP5
FDAT_ACT= FPlace_R1_L6_S2_NP5
BAS(#PTP_PARAMS,100)
PTP XPlace_R1_L6_S2_NP5 C_DIS
;ENDFOLD
TRIGGER WHEN DISTANCE=1 DELAY=-1 DO Schrittmerker_R1Place(10658,10659,FPlace_R1_L6_S2_NP6,XPlace_R1_L6_S2_NP6) PRIO=-1
;FOLD PTP Place_R1_L6_S2_NP6 CONT Vel=100 % PPlace_R1_L6_S2_NP6 Tool[1]:Upper Gripper Base[0];%{PE}%R8.3.21,%MKUKATPBASIS,%CMOVE,%VPTP,%P 1:PTP, 2:Place_R1_L6_S2_NP6, 3:C_DIS, 5:100, 7:PPlace_R1_L6_S2_NP6
$BWDSTART=FALSE
PDAT_ACT= PPPlace_R1_L6_S2_NP6
FDAT_ACT= FPlace_R1_L6_S2_NP6
BAS(#PTP_PARAMS,100)
PTP XPlace_R1_L6_S2_NP6 C_DIS
;ENDFOLD

TRIGGER WHEN DISTANCE=1 DELAY=-1 DO Schrittmerker_R1Place(10659,10501,FHOME,$nullframe,XHOME) PRIO=-1
;FOLD PTP HOME Vel=100 % PHome;%{PE}%R8.3.21,%MKUKATPBASIS,%CMOVE,%VPTP,%P 1:PTP, 2:HOME, 3:, 5:100, 7:PHome
$BWDSTART=FALSE
PDAT_ACT= PPHome
FDAT_ACT= FHOME
BAS(#PTP_PARAMS,100)
PTP XHOME
;ENDFOLD

;***************************************************
;FOLD Final tasks.
; Robot out of area Rack 1 Level 6
RobAusStorage1_6_A72=RESET_IN_AREA
;***************************************************
; stop cyclic clearence check
$CYCFLAG[ciFreigabeSPS]=DISABLE_MONITORING
;***************************************************
; Disable collision detection
;FOLD COLLDETECT Off ;%{PE}
;FOLD Parameters ;%{h}
;Params IlfProvider=kukaroboter.basistech.inlineforms.colldetect.off; CollDetect.Command=Off
;ENDFOLD
USE_CD_PARAMS(0)
;ENDFOLD
;***************************************************
;ENDFOLD
;***************************************************

END

; ##################################################

GLOBAL DEF UP_Place_R1_L6_S3( )
;***************************************************
; Place part on:
;    Rack  1
;    Level 6
;    Shelf 3
;***************************************************
;FOLD Preconditions - Vorraussetzungen
;***************************************************
; Enable collision detection
;FOLD COLLDETECT SetLimits Axis1: 150 % Axis2: 200 % Axis3: 150 % Axis4: 200 % Axis5: 150 % Axis6: 150 % ;%{PE}
;FOLD Parameters ;%{h}
;Params IlfProvider=kukaroboter.basistech.inlineforms.colldetect.setlimits; CollDetect.Command=SetLimits; CollDetect.Axis1=150; CollDetect.Axis2=200; CollDetect.Axis3=150; CollDetect.Axis4=200; CollDetect.Axis5=150; CollDetect.Axis6=150
;ENDFOLD
SET_TQ_VALUES(150, 200, 150, 200, 150, 150)
;ENDFOLD
;***************************************************
; Check for part in gripper (tool 1).
CheckPartPresent(OCCUPIED_GRIPPER,PART_ON_TOOL_1)
;***************************************************
; Enable part lost detection for tool 1
SetPartLostDetection(PART_ON_TOOL_1)
;***************************************************
; Set load data.
SetLoadData( )
;***************************************************
; Robot has to start from home position.
IF NOT $IN_HOME THEN
  UP_HomeToHome(0)
ENDIF
;***************************************************
;ENDFOLD

TRIGGER WHEN DISTANCE=1 DELAY=-1 DO Schrittmerker_R1Place(10501,10501,FHOME,$nullframe,XHOME) PRIO=-1
;FOLD PTP HOME Vel=12 % PHome;%{PE}%R8.3.21,%MKUKATPBASIS,%CMOVE,%VPTP,%P 1:PTP, 2:HOME, 3:, 5:12, 7:PHome
$BWDSTART=FALSE
PDAT_ACT= PPHome
FDAT_ACT= FHOME
BAS(#PTP_PARAMS,12)
PTP XHOME
;ENDFOLD

;***************************************************
;FOLD Area clearence handshake.
IF NOT $FLAG[M_Inbetriebnahme] THEN
  ;-------------------------------------------------
  ; Request area clearence.
  AnfStoer_Store1_6_A104=SET_REQUEST
  ;-------------------------------------------------
  ; Wait for area clearence from PLC.
  WAIT_FOR_INPUT("Frg_Storage1_6_E72",TRUE)
  ;-------------------------------------------------
  ; Reset area clearence request.
  AnfStoer_Store1_6_A104=RESET_REQUEST
  ;-------------------------------------------------
  ; start cyclic clearence check
  $CYCFLAG[ciFreigabeSPS]=Frg_Storage1_6_E72
  ;-------------------------------------------------
ENDIF
;***************************************************
; set "robot in area"
RobAusStorage1_6_A72=SET_IN_AREA
;ENDFOLD
;***************************************************

;***************************************************
;FOLD Check for Teachmode
IF $FLAG[M_Teachen] THEN
  WAIT FOR $T1
ENDIF
;ENDFOLD
;***************************************************

; move to the rack
TRIGGER WHEN DISTANCE=1 DELAY=-1 DO Schrittmerker_R1Place(10670,10501,FPlace_R1_L6_S3_VP1,XPlace_R1_L6_S3_VP1) PRIO=-1
;FOLD PTP Place_R1_L6_S3_VP1 CONT Vel=12 % PPlace_R1_L6_S3_VP1 Tool[1]:Upper Gripper Base[0];%{PE}%R8.3.21,%MKUKATPBASIS,%CMOVE,%VPTP,%P 1:PTP, 2:Place_R1_L6_S3_VP1, 3:C_DIS, 5:12, 7:PPlace_R1_L6_S3_VP1
$BWDSTART=FALSE
PDAT_ACT= PPPlace_R1_L6_S3_VP1
FDAT_ACT= FPlace_R1_L6_S3_VP1
BAS(#PTP_PARAMS,12)
PTP XPlace_R1_L6_S3_VP1 C_DIS
;ENDFOLD
TRIGGER WHEN DISTANCE=1 DELAY=-1 DO Schrittmerker_R1Place(10671,10670,FPlace_R1_L6_S3_VP2,XPlace_R1_L6_S3_VP2) PRIO=-1
;FOLD PTP Place_R1_L6_S3_VP2 CONT Vel=12 % PPlace_R1_L6_S3_VP2 Tool[1]:Upper Gripper Base[0];%{PE}%R8.3.21,%MKUKATPBASIS,%CMOVE,%VPTP,%P 1:PTP, 2:Place_R1_L6_S3_VP2, 3:C_DIS, 5:12, 7:PPlace_R1_L6_S3_VP2
$BWDSTART=FALSE
PDAT_ACT= PPPlace_R1_L6_S3_VP2
FDAT_ACT= FPlace_R1_L6_S3_VP2
BAS(#PTP_PARAMS,12)
PTP XPlace_R1_L6_S3_VP2 C_DIS
;ENDFOLD

TRIGGER WHEN DISTANCE=1 DELAY=-1 DO Schrittmerker_R1Place(10672,10671,FPlace_R1_L6_S3_Check,XPlace_R1_L6_S3_Check) PRIO=-1
;FOLD PTP Place_R1_L6_S3_Check Vel=12 % PPlace_R1_L6_S3_Check Tool[1]:Upper Gripper Base[1]:Rack1;%{PE}%R8.3.21,%MKUKATPBASIS,%CMOVE,%VPTP,%P 1:PTP, 2:Place_R1_L6_S3_Check, 3:, 5:12, 7:PPlace_R1_L6_S3_Check
$BWDSTART=FALSE
PDAT_ACT= PPPlace_R1_L6_S3_Check
FDAT_ACT= FPlace_R1_L6_S3_Check
BAS(#PTP_PARAMS,12)
PTP XPlace_R1_L6_S3_Check
;ENDFOLD

;***************************************************
;FOLD Pruefe Platz frei
IF (DetectPart(CHECK_SHELF,PLACE)==OCCUPIED) THEN
  UP_Rueckzug_R1Place( )
  RETURN
ENDIF
;ENDFOLD
;***************************************************

TRIGGER WHEN DISTANCE=1 DELAY=-1 DO Schrittmerker_R1Place(10673,10672,FPlace_R1_L6_S3_VP3,XPlace_R1_L6_S3_VP3) PRIO=-1
;FOLD LIN Place_R1_L6_S3_VP3 CONT Vel=0.5 m/s LPlace_R1_L6_S3_VP3 Tool[1]:Upper Gripper Base[1]:Rack1;%{PE}%R8.3.21,%MKUKATPBASIS,%CMOVE,%VLIN,%P 1:LIN, 2:Place_R1_L6_S3_VP3, 3:C_DIS C_DIS, 5:0.5, 7:LPlace_R1_L6_S3_VP3
$BWDSTART=FALSE
LDAT_ACT= LLPlace_R1_L6_S3_VP3
FDAT_ACT= FPlace_R1_L6_S3_VP3
BAS(#CP_PARAMS,0.5)
LIN XPlace_R1_L6_S3_VP3 C_DIS C_DIS
;ENDFOLD
TRIGGER WHEN DISTANCE=1 DELAY=-1 DO Schrittmerker_R1Place(10674,10673,FPlace_R1_L6_S3_VP4,XPlace_R1_L6_S3_VP4) PRIO=-1
;FOLD LIN Place_R1_L6_S3_VP4 CONT Vel=0.5 m/s LPlace_R1_L6_S3_VP4 Tool[1]:Upper Gripper Base[1]:Rack1;%{PE}%R8.3.21,%MKUKATPBASIS,%CMOVE,%VLIN,%P 1:LIN, 2:Place_R1_L6_S3_VP4, 3:C_DIS C_DIS, 5:0.5, 7:LPlace_R1_L6_S3_VP4
$BWDSTART=FALSE
LDAT_ACT= LLPlace_R1_L6_S3_VP4
FDAT_ACT= FPlace_R1_L6_S3_VP4
BAS(#CP_PARAMS,0.5)
LIN XPlace_R1_L6_S3_VP4 C_DIS C_DIS
;ENDFOLD
TRIGGER WHEN DISTANCE=1 DELAY=-1 DO Schrittmerker_R1Place(10675,10674,FPlace_R1_L6_S3_VP5,XPlace_R1_L6_S3_VP5) PRIO=-1
;FOLD LIN Place_R1_L6_S3_VP5 CONT Vel=0.5 m/s LPlace_R1_L6_S3_VP5 Tool[1]:Upper Gripper Base[1]:Rack1;%{PE}%R8.3.21,%MKUKATPBASIS,%CMOVE,%VLIN,%P 1:LIN, 2:Place_R1_L6_S3_VP5, 3:C_DIS C_DIS, 5:0.5, 7:LPlace_R1_L6_S3_VP5
$BWDSTART=FALSE
LDAT_ACT= LLPlace_R1_L6_S3_VP5
FDAT_ACT= FPlace_R1_L6_S3_VP5
BAS(#CP_PARAMS,0.5)
LIN XPlace_R1_L6_S3_VP5 C_DIS C_DIS
;ENDFOLD

;FOLD Test the way back home - part 1
CONTINUE
IF ($FLAG[M_Test_GrdstFahren1] AND NOT $FLAG[M_Test_GrdstFahren2]) THEN
  $FLAG[M_Test_GrdstFahren2]=TRUE
  UP_Rueckzug( )
  RETURN
ENDIF
;ENDFOLD

;-------------------------------
; Place part position
;-------------------------------
TRIGGER WHEN DISTANCE=1 DELAY=-1 DO Schrittmerker_R1Place(10676,10677,FPlace_R1_L6_S3_AP,XPlace_R1_L6_S3_AP) PRIO=-1
;FOLD LIN Place_R1_L6_S3_AP Vel=0.2 m/s LPlace_R1_L6_S3_AP Tool[1]:Upper Gripper Base[1]:Rack1;%{PE}%R8.3.21,%MKUKATPBASIS,%CMOVE,%VLIN,%P 1:LIN, 2:Place_R1_L6_S3_AP, 3:, 5:0.2, 7:LPlace_R1_L6_S3_AP
$BWDSTART=FALSE
LDAT_ACT= LLPlace_R1_L6_S3_AP
FDAT_ACT= FPlace_R1_L6_S3_AP
BAS(#CP_PARAMS,0.2)
LIN XPlace_R1_L6_S3_AP
;ENDFOLD

;FOLD Test the way back home - part 2
CONTINUE
IF $FLAG[M_Test_GrdstFahren2] THEN
  $FLAG[M_Test_GrdstFahren2]=FALSE
  UP_Rueckzug( )
  RETURN
ENDIF
;ENDFOLD

;***************************************************
; Disable part lost detection
SetPartLostDetection(NO_PART)
;***************************************************

TRIGGER WHEN DISTANCE=1 DELAY=-1 DO Schrittmerker_R1Place(10677,10678,FPlace_R1_L6_S3_NP1,XPlace_R1_L6_S3_NP1) PRIO=-1
;FOLD LIN Place_R1_L6_S3_NP1 Vel=0.2 m/s LPlace_R1_L6_S3_NP1 Tool[1]:Upper Gripper Base[1]:Rack1;%{PE}%R8.3.21,%MKUKATPBASIS,%CMOVE,%VLIN,%P 1:LIN, 2:Place_R1_L6_S3_NP1, 3:C_DIS C_DIS, 5:0.2, 7:LPlace_R1_L6_S3_NP1
$BWDSTART=FALSE
LDAT_ACT= LLPlace_R1_L6_S3_NP1
FDAT_ACT= FPlace_R1_L6_S3_NP1
BAS(#CP_PARAMS,0.2)
LIN XPlace_R1_L6_S3_NP1
;ENDFOLD

;***************************************************
; Check for part present (empty gripper)
CheckPartPresent(EMPTY_GRIPPER)
;***************************************************
; set load data
SetLoadData( )
;***************************************************

TRIGGER WHEN DISTANCE=1 DELAY=-1 DO Schrittmerker_R1Place(10678,10679,FPlace_R1_L6_S3_NP2,XPlace_R1_L6_S3_NP2) PRIO=-1
;FOLD LIN Place_R1_L6_S3_NP2 CONT Vel=0.5 m/s LPlace_R1_L6_S3_NP2 Tool[1]:Upper Gripper Base[1]:Rack1;%{PE}%R8.3.21,%MKUKATPBASIS,%CMOVE,%VLIN,%P 1:LIN, 2:Place_R1_L6_S3_NP2, 3:C_DIS C_DIS, 5:0.5, 7:LPlace_R1_L6_S3_NP2
$BWDSTART=FALSE
LDAT_ACT= LLPlace_R1_L6_S3_NP2
FDAT_ACT= FPlace_R1_L6_S3_NP2
BAS(#CP_PARAMS,0.5)
LIN XPlace_R1_L6_S3_NP2 C_DIS C_DIS
;ENDFOLD
TRIGGER WHEN DISTANCE=1 DELAY=-1 DO Schrittmerker_R1Place(10679,10680,FPlace_R1_L6_S3_NP3,XPlace_R1_L6_S3_NP3) PRIO=-1
;FOLD LIN Place_R1_L6_S3_NP3 Vel=0.5 m/s LPlace_R1_L6_S3_NP3 Tool[1]:Upper Gripper Base[1]:Rack1;%{PE}%R8.3.21,%MKUKATPBASIS,%CMOVE,%VLIN,%P 1:LIN, 2:Place_R1_L6_S3_NP3, 3:, 5:0.5, 7:LPlace_R1_L6_S3_NP3
$BWDSTART=FALSE
LDAT_ACT= LLPlace_R1_L6_S3_NP3
FDAT_ACT= FPlace_R1_L6_S3_NP3
BAS(#CP_PARAMS,0.5)
LIN XPlace_R1_L6_S3_NP3
;ENDFOLD
TRIGGER WHEN DISTANCE=1 DELAY=-1 DO Schrittmerker_R1Place(10680,10681,FPlace_R1_L6_S3_NP4,XPlace_R1_L6_S3_NP4) PRIO=-1
;FOLD PTP Place_R1_L6_S3_NP4 CONT Vel=100 % PPlace_R1_L6_S3_NP4 Tool[1]:Upper Gripper Base[0];%{PE}%R8.3.21,%MKUKATPBASIS,%CMOVE,%VPTP,%P 1:PTP, 2:Place_R1_L6_S3_NP4, 3:C_DIS, 5:100, 7:PPlace_R1_L6_S3_NP4
$BWDSTART=FALSE
PDAT_ACT= PPPlace_R1_L6_S3_NP4
FDAT_ACT= FPlace_R1_L6_S3_NP4
BAS(#PTP_PARAMS,100)
PTP XPlace_R1_L6_S3_NP4 C_DIS
;ENDFOLD
TRIGGER WHEN DISTANCE=1 DELAY=-1 DO Schrittmerker_R1Place(10681,10682,FPlace_R1_L6_S3_NP5,XPlace_R1_L6_S3_NP5) PRIO=-1
;FOLD PTP Place_R1_L6_S3_NP5 CONT Vel=100 % PPlace_R1_L6_S3_NP5 Tool[1]:Upper Gripper Base[0];%{PE}%R8.3.21,%MKUKATPBASIS,%CMOVE,%VPTP,%P 1:PTP, 2:Place_R1_L6_S3_NP5, 3:C_DIS, 5:100, 7:PPlace_R1_L6_S3_NP5
$BWDSTART=FALSE
PDAT_ACT= PPPlace_R1_L6_S3_NP5
FDAT_ACT= FPlace_R1_L6_S3_NP5
BAS(#PTP_PARAMS,100)
PTP XPlace_R1_L6_S3_NP5 C_DIS
;ENDFOLD
TRIGGER WHEN DISTANCE=1 DELAY=-1 DO Schrittmerker_R1Place(10682,10683,FPlace_R1_L6_S3_NP6,XPlace_R1_L6_S3_NP6) PRIO=-1
;FOLD PTP Place_R1_L6_S3_NP6 CONT Vel=100 % PPlace_R1_L6_S3_NP6 Tool[1]:Upper Gripper Base[0];%{PE}%R8.3.21,%MKUKATPBASIS,%CMOVE,%VPTP,%P 1:PTP, 2:Place_R1_L6_S3_NP6, 3:C_DIS, 5:100, 7:PPlace_R1_L6_S3_NP6
$BWDSTART=FALSE
PDAT_ACT= PPPlace_R1_L6_S3_NP6
FDAT_ACT= FPlace_R1_L6_S3_NP6
BAS(#PTP_PARAMS,100)
PTP XPlace_R1_L6_S3_NP6 C_DIS
;ENDFOLD

TRIGGER WHEN DISTANCE=1 DELAY=-1 DO Schrittmerker_R1Place(10683,10501,FHOME,$nullframe,XHOME) PRIO=-1
;FOLD PTP HOME Vel=100 % PHome;%{PE}%R8.3.21,%MKUKATPBASIS,%CMOVE,%VPTP,%P 1:PTP, 2:HOME, 3:, 5:100, 7:PHome
$BWDSTART=FALSE
PDAT_ACT= PPHome
FDAT_ACT= FHOME
BAS(#PTP_PARAMS,100)
PTP XHOME
;ENDFOLD

;***************************************************
;FOLD Final tasks.
; Robot out of area Rack 1 Level 6
RobAusStorage1_6_A72=RESET_IN_AREA
;***************************************************
; stop cyclic clearence check
$CYCFLAG[ciFreigabeSPS]=DISABLE_MONITORING
;***************************************************
; Disable collision detection
;FOLD COLLDETECT Off ;%{PE}
;FOLD Parameters ;%{h}
;Params IlfProvider=kukaroboter.basistech.inlineforms.colldetect.off; CollDetect.Command=Off
;ENDFOLD
USE_CD_PARAMS(0)
;ENDFOLD
;***************************************************
;ENDFOLD
;***************************************************

END

; ##################################################

GLOBAL DEF UP_Place_R1_L6_S4( )
;***************************************************
; Place part on:
;    Rack  1
;    Level 6
;    Shelf 4
;***************************************************
;FOLD Preconditions - Vorraussetzungen
;***************************************************
; Enable collision detection
;FOLD COLLDETECT SetLimits Axis1: 150 % Axis2: 200 % Axis3: 150 % Axis4: 200 % Axis5: 150 % Axis6: 150 % ;%{PE}
;FOLD Parameters ;%{h}
;Params IlfProvider=kukaroboter.basistech.inlineforms.colldetect.setlimits; CollDetect.Command=SetLimits; CollDetect.Axis1=150; CollDetect.Axis2=200; CollDetect.Axis3=150; CollDetect.Axis4=200; CollDetect.Axis5=150; CollDetect.Axis6=150
;ENDFOLD
SET_TQ_VALUES(150, 200, 150, 200, 150, 150)
;ENDFOLD
;***************************************************
; Check for part in gripper (tool 1).
CheckPartPresent(OCCUPIED_GRIPPER,PART_ON_TOOL_1)
;***************************************************
; Enable part lost detection for tool 1
SetPartLostDetection(PART_ON_TOOL_1)
;***************************************************
; Set load data.
SetLoadData( )
;***************************************************
; Robot has to start from home position.
IF NOT $IN_HOME THEN
  UP_HomeToHome(0)
ENDIF
;***************************************************
;ENDFOLD

TRIGGER WHEN DISTANCE=1 DELAY=-1 DO Schrittmerker_R1Place(10501,10501,FHOME,$nullframe,XHOME) PRIO=-1
;FOLD PTP HOME Vel=12 % PHome;%{PE}%R8.3.21,%MKUKATPBASIS,%CMOVE,%VPTP,%P 1:PTP, 2:HOME, 3:, 5:12, 7:PHome
$BWDSTART=FALSE
PDAT_ACT= PPHome
FDAT_ACT= FHOME
BAS(#PTP_PARAMS,12)
PTP XHOME
;ENDFOLD

;***************************************************
;FOLD Area clearence handshake.
IF NOT $FLAG[M_Inbetriebnahme] THEN
  ;-------------------------------------------------
  ; Request area clearence.
  AnfStoer_Store1_6_A104=SET_REQUEST
  ;-------------------------------------------------
  ; Wait for area clearence from PLC.
  WAIT_FOR_INPUT("Frg_Storage1_6_E72",TRUE)
  ;-------------------------------------------------
  ; Reset area clearence request.
  AnfStoer_Store1_6_A104=RESET_REQUEST
  ;-------------------------------------------------
  ; start cyclic clearence check
  $CYCFLAG[ciFreigabeSPS]=Frg_Storage1_6_E72
  ;-------------------------------------------------
ENDIF
;***************************************************
; set "robot in area"
RobAusStorage1_6_A72=SET_IN_AREA
;ENDFOLD
;***************************************************

;***************************************************
;FOLD Check for Teachmode
IF $FLAG[M_Teachen] THEN
  WAIT FOR $T1
ENDIF
;ENDFOLD
;***************************************************

; move to the rack
TRIGGER WHEN DISTANCE=1 DELAY=-1 DO Schrittmerker_R1Place(10690,10501,FPlace_R1_L6_S4_VP1,XPlace_R1_L6_S4_VP1) PRIO=-1
;FOLD PTP Place_R1_L6_S4_VP1 CONT Vel=12 % PPlace_R1_L6_S4_VP1 Tool[1]:Upper Gripper Base[0];%{PE}%R8.3.21,%MKUKATPBASIS,%CMOVE,%VPTP,%P 1:PTP, 2:Place_R1_L6_S4_VP1, 3:C_DIS, 5:12, 7:PPlace_R1_L6_S4_VP1
$BWDSTART=FALSE
PDAT_ACT= PPPlace_R1_L6_S4_VP1
FDAT_ACT= FPlace_R1_L6_S4_VP1
BAS(#PTP_PARAMS,12)
PTP XPlace_R1_L6_S4_VP1 C_DIS
;ENDFOLD
TRIGGER WHEN DISTANCE=1 DELAY=-1 DO Schrittmerker_R1Place(10691,10690,FPlace_R1_L6_S4_VP2,XPlace_R1_L6_S4_VP2) PRIO=-1
;FOLD PTP Place_R1_L6_S4_VP2 CONT Vel=12 % PPlace_R1_L6_S4_VP2 Tool[1]:Upper Gripper Base[0];%{PE}%R8.3.21,%MKUKATPBASIS,%CMOVE,%VPTP,%P 1:PTP, 2:Place_R1_L6_S4_VP2, 3:C_DIS, 5:12, 7:PPlace_R1_L6_S4_VP2
$BWDSTART=FALSE
PDAT_ACT= PPPlace_R1_L6_S4_VP2
FDAT_ACT= FPlace_R1_L6_S4_VP2
BAS(#PTP_PARAMS,12)
PTP XPlace_R1_L6_S4_VP2 C_DIS
;ENDFOLD

